// TwinCAT 3 PLC project tcl_BaseClasses
// Title: tcl_BaseClasses
// Company: Red Rock Controls Limited
// Author: Roger Christopher
// ProjectVersion: 1.1.70.0
// Description: ResultAggregate updated to use array of I_ExecutionResult interfaces for transparency during debugging
// ProgramVersion: 3.1.4023.0
// CompilerDefines: VISU_USEPROPERTYINFO
// libraries:
//   Tc2_Standard, * (Beckhoff Automation GmbH)
//   Tc2_System, * (Beckhoff Automation GmbH)
//   Tc2_Utilities, * (Beckhoff Automation GmbH)
//   Tc3_DynamicMemory, * (Beckhoff Automation GmbH)
//   Tc3_EventLogger, * (Beckhoff Automation GmbH)
//   Tc3_Module, * (Beckhoff Automation GmbH)
//   tcl_StringUtils, * (Red Rock Controls Limited)
// project tree:
//   Classes/Change Monitoring/ T_Monitor_INT.TcPOU, T_Monitor_DINT.TcPOU, T_Monitor_Structure.TcPOU
//   Classes/Execution Result Aggregate/ T_ResultAggregate.TcPOU
//   Classes/Execution/Execution/ I_Execution.TcIO, I_ExecutionResult.TcIO, T_Execution.TcPOU, T_ExecutionState.TcDUT
//   Classes/Function Block Wrappers/Classes/ T_Counter.TcPOU, T_FallingEdge.TcPOU, T_MonitoredValue.TcPOU, T_OffTimer.TcPOU, T_OnTimer.TcPOU, T_PulseTimer.TcPOU, T_RisingEdge.TcPOU, T_SquareWave.TcPOU, T_StructureCrcMonitor.TcPOU, T_ValueMonitor.TcPOU, T_ValueMonitorEx.TcPOU
//   Classes/List Of Interfaces/ I_ListItem.TcIO, I_ListOfInterfaces.TcIO, T_ListOfInterfaces.TcPOU
//   Classes/Logger/ I_Logger.TcIO, T_Logger.TcPOU, T_Message.TcPOU
//   Classes/Notifications/List Of Handlers/ T_ListONotificationHandlers.TcPOU
//   Classes/Notifications/Notification Handler/ I_NotificationHandler.TcIO, T_NotificationHandler.TcPOU
//   Classes/Notifications/Notification/ I_Notification.TcIO, T_Notification.TcPOU
//   Classes/Nullable Base Class/ T_NullableBaseClass.TcPOU
//   Classes/Object base class/ T_Object.TcPOU
//   Classes/Stream/ E_ArgTypeId.TcDUT, I_StreamReader.TcIO, I_StreamWriter.TcIO, T_Stream.TcPOU
//   Functions/ F_CompareMem.TcPOU, F_CopyMem.TcPOU, F_DetectOnlineChange.TcPOU, F_DINT_TO_UDINT.TcPOU, F_Dec.TcPOU, F_InLimits.TcPOU, F_ErrorIdToString.TcPOU, F_Inc.TcPOU, F_LinearInterpolation.TcPOU, F_LogError.TcPOU, F_LogMessage.TcPOU, F_LogWarning.TcPOU, F_ReadFlag.TcPOU, F_TaskTime.TcPOU, F_NotEqual.TcPOU, F_Toggle.TcPOU, F_UDINT_TO_DINT.TcPOU, F_ClearMem.TcPOU, F_Equals.TcPOU, F_GetAdsPort.TcPOU
//   / Globals.TcGVL
//   Version/ Global_Version.TcGVL
// real-time tasks:
//   TASK PlcTask: cycle T#10ms, priority 20, ADS port 350
//   TASK PlcTask1: cycle T#10ms, priority 21, ADS port 351

// ---- Classes/Execution/Execution/T_ExecutionState.TcDUT
{attribute 'qualified_only'}
{attribute 'strict'}
TYPE
    T_ExecutionState :
    (
        Ready := 0,
        Starting,
        Busy
    );
END_TYPE

// ---- Classes/Stream/E_ArgTypeId.TcDUT
{attribute 'qualified_only'}
TYPE
    E_ArgTypeId :
    (
        Unknown := 0,
        Type_Blob,
        Type_BOOL,
        Type_BYTE,
        Type_DINT,
        Type_INT,
        Type_LINT,
        Type_LREAL,
        Type_PVOID,
        Type_REAL,
        Type_STRING,
        Type_UDINT,
        Type_UINT,
        Type_ULINT,
        MaxSupportType
    );
END_TYPE

// ---- Globals.TcGVL
VAR_GLOBAL
	DefaultLogger : T_Logger;
END_VAR

// ---- Version/Global_Version.TcGVL
{attribute 'TcGenerated'}
{attribute 'no-analysis'}
{attribute 'linkalways'}
// This function has been automatically generated from the project information.
VAR_GLOBAL CONSTANT
	{attribute 'const_non_replaced'}
	stLibVersion_tcl_BaseClasses : ST_LibVersion := (iMajor := 1, iMinor := 1, iBuild := 70, iRevision := 0, nFlags := 0, sVersion := '1.1.70.0');
END_VAR

// ---- Classes/Execution/Execution/I_Execution.TcIO
INTERFACE I_Execution

METHOD Abort
VAR_INPUT
END_VAR
END_METHOD

PROPERTY Aborted : BOOL
GET
END_GET
END_PROPERTY

PROPERTY Busy : BOOL
GET
END_GET
END_PROPERTY

METHOD Clear
VAR_INPUT
END_VAR
END_METHOD

PROPERTY Done : BOOL
GET
END_GET
END_PROPERTY

PROPERTY Error : BOOL
GET
END_GET
END_PROPERTY

PROPERTY ErrorMsg : T_MaxString
GET
END_GET
END_PROPERTY

PROPERTY Ready : BOOL
GET
END_GET
END_PROPERTY

METHOD Start : I_ExecutionResult;
VAR_INPUT
END_VAR
END_METHOD

PROPERTY Starting : BOOL
GET
END_GET
END_PROPERTY

END_INTERFACE

// ---- Classes/Execution/Execution/I_ExecutionResult.TcIO
INTERFACE I_ExecutionResult EXTENDS I_ListItem // Just exposes the state of the execution object. Usage is "Result := Execution.Start()" so Result can be monitored

METHOD Abort
VAR_INPUT
END_VAR
END_METHOD

PROPERTY Aborted : BOOL
GET
END_GET
END_PROPERTY

PROPERTY Aborting : BOOL
GET
END_GET
END_PROPERTY

PROPERTY Busy : BOOL
GET
END_GET
END_PROPERTY

METHOD Clear
END_METHOD

PROPERTY Done : BOOL
GET
END_GET
END_PROPERTY

PROPERTY Error : BOOL
GET
END_GET
END_PROPERTY

PROPERTY ErrorMsg : T_MaxString
GET
END_GET
END_PROPERTY

PROPERTY Ready : BOOL
GET
END_GET
END_PROPERTY

PROPERTY Starting : BOOL
GET
END_GET
END_PROPERTY

END_INTERFACE

// ---- Classes/List Of Interfaces/I_ListItem.TcIO
INTERFACE I_ListItem EXTENDS __SYSTEM.IQueryInterface

END_INTERFACE

// ---- Classes/List Of Interfaces/I_ListOfInterfaces.TcIO
INTERFACE I_ListOfInterfaces EXTENDS I_ListItem

METHOD AddInterface
VAR_INPUT
    InterfacePointer : I_ListItem;
END_VAR
END_METHOD

PROPERTY Count : DINT
GET
END_GET
END_PROPERTY

METHOD GetInterface : I_ListItem
VAR_INPUT
    Index : DINT;
END_VAR
END_METHOD

END_INTERFACE

// ---- Classes/Logger/I_Logger.TcIO
INTERFACE I_Logger

METHOD LogCritical
VAR_INPUT
	Source	: I_TcSourceInfo;
    Message : T_MaxString;
END_VAR
END_METHOD

METHOD LogDebug
VAR_INPUT
	Source	: I_TcSourceInfo;
    Message : T_MaxString;
END_VAR
END_METHOD

METHOD LogError
VAR_INPUT
	Source	: I_TcSourceInfo;
    Message : T_MaxString;
END_VAR
END_METHOD

METHOD LogInfo
VAR_INPUT
	Source	: I_TcSourceInfo;
    Message : T_MaxString;
END_VAR
END_METHOD

METHOD LogWarning
VAR_INPUT
	Source	: I_TcSourceInfo;
    Message : T_MaxString;
END_VAR
END_METHOD

END_INTERFACE

// ---- Classes/Notifications/Notification Handler/I_NotificationHandler.TcIO
{attribute 'hide'}
INTERFACE I_NotificationHandler EXTENDS __SYSTEM.IQueryInterface

PROPERTY Args : I_StreamReader
GET
END_GET
END_PROPERTY

PROPERTY NotificationCount : DINT
GET
END_GET
END_PROPERTY

METHOD RaiseNotification
VAR_INPUT
    NotificationArgs : I_StreamReader;
END_VAR
END_METHOD

END_INTERFACE

// ---- Classes/Notifications/Notification/I_Notification.TcIO
INTERFACE I_Notification

METHOD AddNotificationHandler : I_Notification
VAR_INPUT
    Handler : I_NotificationHandler;
END_VAR
END_METHOD

PROPERTY Args : I_StreamWriter
GET
END_GET
END_PROPERTY

METHOD ClearNotificationHandlers : I_Notification
VAR_INPUT
END_VAR
END_METHOD

METHOD Raise
END_METHOD

END_INTERFACE

// ---- Classes/Stream/I_StreamReader.TcIO
INTERFACE I_StreamReader

{attribute 'monitoring' := 'call'}
PROPERTY BufferAddress : PVOID
GET
END_GET
END_PROPERTY

METHOD GetNextArgTypeId : E_ArgTypeId
END_METHOD

METHOD Read_BLOB
VAR_INPUT
    BlobToCopyTo : ANY;
END_VAR
END_METHOD

METHOD Read_BOOL : BOOL
END_METHOD

METHOD Read_BYTE : BYTE
END_METHOD

METHOD Read_DATA
VAR_INPUT
    DataAddress : PVOID;
    DataLength  : UDINT;
END_VAR
END_METHOD

METHOD Read_DINT : DINT
END_METHOD

METHOD Read_INT : INT
END_METHOD

METHOD Read_LINT : LINT
END_METHOD

METHOD Read_LREAL : LREAL
END_METHOD

METHOD Read_PVOID : PVOID
END_METHOD

METHOD Read_REAL : REAL
END_METHOD

METHOD Read_STRING : STRING(255)
END_METHOD

METHOD Read_STRUCT
VAR_INPUT
    StructureAddress : PVOID;
    StructureLength  : UDINT;
END_VAR
END_METHOD

METHOD Read_UDINT : UDINT
END_METHOD

METHOD Read_UINT : UINT
END_METHOD

METHOD Read_ULINT : ULINT
END_METHOD

{attribute 'monitoring' := 'call'}
PROPERTY ReadPosition : UDINT
GET
END_GET
END_PROPERTY

METHOD SetReadPosition : I_StreamWriter
VAR_INPUT
    Position : UDINT;
END_VAR
END_METHOD

{attribute 'monitoring' := 'call'}
PROPERTY StreamLength : UDINT
GET
END_GET
END_PROPERTY

{attribute 'monitoring' := 'call'}
PROPERTY WritePosition : UDINT
GET
END_GET
END_PROPERTY

END_INTERFACE

// ---- Classes/Stream/I_StreamWriter.TcIO
INTERFACE I_StreamWriter

METHOD Add_BLOB : I_StreamWriter
VAR_INPUT
    BlobToCopyFrom : ANY;
END_VAR
END_METHOD

METHOD Add_BOOL : I_StreamWriter
VAR_INPUT
    Value : BOOL;
END_VAR
END_METHOD

METHOD Add_BYTE : I_StreamWriter
VAR_INPUT
    Value : BYTE;
END_VAR
END_METHOD

METHOD Add_DATA : I_StreamWriter
VAR_INPUT
    DataAddress : PVOID;
    DataLength  : UDINT;
END_VAR
END_METHOD

METHOD Add_DINT : I_StreamWriter
VAR_INPUT
    Value : DINT;
END_VAR
END_METHOD

METHOD Add_INT : I_StreamWriter
VAR_INPUT
    Value : INT;
END_VAR
END_METHOD

METHOD Add_LINT : I_StreamWriter
VAR_INPUT
    Value : LINT;
END_VAR
END_METHOD

METHOD Add_LREAL : I_StreamWriter
VAR_INPUT
    Value : LREAL;
END_VAR
END_METHOD

METHOD Add_PVOID : I_StreamWriter
VAR_INPUT
    Value : PVOID;
END_VAR
END_METHOD

METHOD Add_REAL : I_StreamWriter
VAR_INPUT
    Value : REAL;
END_VAR
END_METHOD

METHOD Add_STRING : I_StreamWriter
VAR_INPUT
    Value : STRING(255);
END_VAR
END_METHOD

METHOD Add_STRUCT : I_StreamWriter
VAR_INPUT
    StructureAddress : PVOID;
    StructureLength  : UDINT;
END_VAR
END_METHOD

METHOD Add_UDINT : I_StreamWriter
VAR_INPUT
    Value : UDINT;
END_VAR
END_METHOD

METHOD Add_UINT : I_StreamWriter
VAR_INPUT
    Value : UINT;
END_VAR
END_METHOD

METHOD Add_ULINT : I_StreamWriter
VAR_INPUT
    Value : ULINT;
END_VAR
END_METHOD

METHOD AppendBytesFromStream
VAR_INPUT
    StreamToAppend        : I_StreamReader;
    NumberOfBytesToAppend : UDINT;
END_VAR
VAR

END_VAR
END_METHOD

{attribute 'monitoring' := 'call'}
PROPERTY BufferAddress : PVOID
GET
END_GET
END_PROPERTY

METHOD Clear : I_StreamWriter
END_METHOD

METHOD Init
VAR_INPUT
    StreamLength : UDINT;
END_VAR
END_METHOD

{attribute 'monitoring' := 'call'}
PROPERTY ReadPosition : UDINT
GET
END_GET
END_PROPERTY

METHOD SetNextArgTypeId : I_StreamWriter
VAR_INPUT
    Value : E_ArgTypeId;
END_VAR
END_METHOD

METHOD SetReadPosition : I_StreamWriter
VAR_INPUT
    Position : UDINT;
END_VAR
END_METHOD

{attribute 'monitoring' := 'call'}
PROPERTY StreamLength : UDINT
GET
END_GET
END_PROPERTY

{attribute 'monitoring' := 'call'}
PROPERTY WritePosition : UDINT
GET
END_GET
END_PROPERTY

END_INTERFACE

// ---- Classes/Logger/T_Logger.TcPOU
{attribute 'no_explicit_call' := 'do not call this POU directly'}
FUNCTION_BLOCK T_Logger IMPLEMENTS I_Logger
VAR
    DebugMessage    : T_Message;
    InfoMessage     : T_Message;
    WarningMessage  : T_Message;
    ErrorMessage    : T_Message;
    CriticalMessage : T_Message;

END_VAR

METHOD LogCritical
VAR_INPUT
	Source	: I_TcSourceInfo;
	Message	: Tc2_System.T_MaxString;
END_VAR
CriticalMessage.Send(TcEventSeverity.Critical, Source,Message);
END_METHOD

METHOD LogDebug
VAR_INPUT
	Source	: I_TcSourceInfo;
	Message	: Tc2_System.T_MaxString;
END_VAR
DebugMessage.Send(TcEventSeverity.Verbose, Source,Message);
END_METHOD

METHOD LogError
VAR_INPUT
	Source	: I_TcSourceInfo;
	Message	: Tc2_System.T_MaxString;
END_VAR
ErrorMessage.Send(TcEventSeverity.Error, Source,Message);
END_METHOD

METHOD LogInfo
VAR_INPUT
	Source	: I_TcSourceInfo;
	Message	: Tc2_System.T_MaxString;
END_VAR
InfoMessage.Send(TcEventSeverity.Info, Source,Message);
END_METHOD

METHOD LogWarning
VAR_INPUT
	Source	: I_TcSourceInfo;
	Message	: Tc2_System.T_MaxString;
END_VAR
WarningMessage.Send(TcEventSeverity.Warning, Source,Message);
END_METHOD

END_FUNCTION_BLOCK

// ---- Classes/Logger/T_Message.TcPOU
FUNCTION_BLOCK T_Message
VAR
    Msg        : FB_TcMessage;
END_VAR

METHOD Send
VAR_INPUT
    Severity : TcEventSeverity;
    Source   : I_TcSourceInfo;
    Message  : Tc2_System.T_MaxString;
END_VAR
VAR
    Result : HRESULT;
END_VAR
CASE Severity OF 
	TcEventSeverity.Critical:
		Result := Msg.CreateEx(TC_EVENTS.PLC_Exceptions.LogCritical, Source);
		
	TcEventSeverity.Error:
		Result := Msg.CreateEx(TC_EVENTS.PLC_Exceptions.LogError, Source);
		
	TcEventSeverity.Warning:
		Result := Msg.CreateEx(TC_EVENTS.PLC_Exceptions.LogWarning, Source);
		
	TcEventSeverity.Info:
		Result := Msg.CreateEx(TC_EVENTS.PLC_Exceptions.LogInfo, Source);
		
	TcEventSeverity.Verbose:
		Result := Msg.CreateEx(TC_EVENTS.PLC_Exceptions.LogDebug, Source);
		
END_CASE

IF Result = S_OK THEN
	Msg.ipArguments.Clear().AddString(Message);
    Msg.Send(0);
	Msg.Release();
ELSE
    F_LogError(Source := 'Logger', 'Failed to create EventLogger.Message instance');
END_IF
END_METHOD

END_FUNCTION_BLOCK

// ---- Functions/F_LogError.TcPOU
FUNCTION F_LogError
VAR_INPUT
    Source  : T_MaxString;
    Message : T_MaxString;
END_VAR
VAR_STAT
    LastMessage        : T_MaxString;
    RepeatMessageCount : UDINT;
END_VAR

IF Message = LastMessage THEN
    F_Inc(RepeatMessageCount);
ELSE
    RepeatMessageCount := 0;
    LastMessage        := Message;
END_IF

IF RepeatMessageCount < 10 THEN // Avoid flooding the Error List...
    ADSLOGSTR(msgCtrlMask := ADSLOG_MSGTYPE_STRING OR ADSLOG_MSGTYPE_ERROR OR ADSLOG_MSGTYPE_LOG,
              msgFmtStr   := CONCAT(Source, ' : %s'),
              strArg      := Message);
END_IF

IF RepeatMessageCount = 10 THEN
    ADSLOGSTR(msgCtrlMask := ADSLOG_MSGTYPE_STRING OR ADSLOG_MSGTYPE_ERROR OR ADSLOG_MSGTYPE_LOG,
              msgFmtStr   := 'Log Errors suspended - too many identical messages!',
              strArg      := '');
END_IF

END_FUNCTION

// ---- Functions/F_Inc.TcPOU
FUNCTION F_Inc : BOOL
VAR_INPUT
    in : ANY_INT;
END_VAR
VAR
    pSINT  : POINTER TO SINT;
    pINT   : POINTER TO INT;
    pDINT  : POINTER TO DINT;
    pLINT  : POINTER TO LINT;
    pUSINT : POINTER TO USINT;
    pUINT  : POINTER TO UINT;
    pUDINT : POINTER TO UDINT;
    pULINT : POINTER TO ULINT;
    pBYTE  : POINTER TO BYTE;
    pWORD  : POINTER TO WORD;
    pDWORD : POINTER TO DWORD;
END_VAR

CASE in.TypeClass OF
    __SYSTEM.TYPE_CLASS.TYPE_SINT:
        pSINT  := in.pValue;
        pSint^ := pSint^ + 1;

    __SYSTEM.TYPE_CLASS.TYPE_INT:
        pINT  := in.pValue;
        pINT^ := pINT^ + 1;

    __SYSTEM.TYPE_CLASS.TYPE_DINT:
        pDINT  := in.pValue;
        pDINT^ := pDINT^ + 1;

    __SYSTEM.TYPE_CLASS.TYPE_LINT:
        pLINT  := in.pValue;
        pLINT^ := pLINT^ + 1;

    __SYSTEM.TYPE_CLASS.TYPE_USINT:
        pUSINT  := in.pValue;
        pUSINT^ := pUSINT^ + 1;

    __SYSTEM.TYPE_CLASS.TYPE_UINT:
        pUINT  := in.pValue;
        pUINT^ := pUINT^ + 1;

    __SYSTEM.TYPE_CLASS.TYPE_UDINT:
        pUDINT  := in.pValue;
        pUDINT^ := pUDINT^ + 1;

    __SYSTEM.TYPE_CLASS.TYPE_ULINT:
        pULINT  := in.pValue;
        pULINT^ := pULINT^ + 1;
		
    __SYSTEM.TYPE_CLASS.TYPE_BYTE:
        pBYTE  := in.pValue;
        pBYTE^ := pBYTE^ + 1;
		
    __SYSTEM.TYPE_CLASS.TYPE_WORD:
        pWORD  := in.pValue;
        pWORD^ := pWORD^ + 1;
		
    __SYSTEM.TYPE_CLASS.TYPE_DWORD:
        pDWORD  := in.pValue;
        pDWORD^ := pDWORD^ + 1;
		
		
END_CASE

END_FUNCTION

// ---- Classes/Change Monitoring/T_Monitor_INT.TcPOU
{attribute 'no_explicit_call':= 'do not call this POU directly'}
FUNCTION_BLOCK T_Monitor_INT
VAR
    _CurrentValue  : INT := UnlikelyValue; 
    _Changed       : BOOL;
END_VAR
VAR CONSTANT
	UnlikelyValue : INT := 12345;
END_VAR

PROPERTY Changed : BOOL
GET
Changed := _Changed;
END_GET
END_PROPERTY

METHOD CyclicUpdate : BOOL
VAR_INPUT
    Value : INT;
END_VAR
_Changed      := Value <> _CurrentValue;
_CurrentValue := Value;
CyclicUpdate  := _Changed;
END_METHOD

METHOD Reset
_CurrentValue := UnlikelyValue;
_Changed      := FALSE;
END_METHOD

END_FUNCTION_BLOCK

// ---- Classes/Change Monitoring/T_Monitor_DINT.TcPOU
{attribute 'no_explicit_call':= 'do not call this POU directly'}
FUNCTION_BLOCK T_Monitor_DINT
VAR
    _CurrentValue  : DINT := UnlikelyValue; 
    _Changed       : BOOL;
END_VAR
VAR CONSTANT
	UnlikelyValue : DINT := 123456789;
END_VAR

PROPERTY Changed : BOOL
GET
Changed := _Changed;
END_GET
END_PROPERTY

METHOD CyclicUpdate : BOOL
VAR_INPUT
    Value : DINT;
END_VAR
_Changed      := Value <> _CurrentValue;
_CurrentValue := Value;
CyclicUpdate  := _Changed;
END_METHOD

METHOD Reset
_CurrentValue := UnlikelyValue;
_Changed      := FALSE;
END_METHOD

END_FUNCTION_BLOCK

// ---- Classes/Change Monitoring/T_Monitor_Structure.TcPOU
{attribute 'no_explicit_call':= 'do not call this POU directly'}
FUNCTION_BLOCK T_Monitor_Structure
VAR
    _Changed   : BOOL;
    Stored_CRC : WORD := 16#FFFF;
END_VAR

PROPERTY Changed : BOOL
GET
Changed := _Changed;
END_GET
END_PROPERTY

METHOD CyclicUpdate : BOOL
VAR_INPUT
    StructureAddress : PVOID;
	StructureLength  : UDINT;
END_VAR
VAR
    CRC : WORD;
END_VAR
CRC := F_DATA_TO_CRC16_CCITT(pData  := StructureAddress,
                             cbData := StructureLength,
                             crc    := 0);
_Changed := (CRC <> Stored_CRC);
IF Changed THEN
    Stored_CRC := CRC;
END_IF
CyclicUpdate := _Changed;
END_METHOD

METHOD Reset
VAR_INPUT
END_VAR
Stored_CRC := 16#FFFF;
_Changed   := FALSE;
END_METHOD

END_FUNCTION_BLOCK

// ---- Classes/Execution Result Aggregate/T_ResultAggregate.TcPOU
FUNCTION_BLOCK T_ResultAggregate IMPLEMENTS I_ExecutionResult
VAR
	Results : ARRAY[0..ResultsUpperBound] OF I_ExecutionResult;
	Count   : UINT;
END_VAR
VAR CONSTANT
	ResultsUpperBound : UINT := 99;
END_VAR

METHOD Abort
VAR
    i      : DINT;
    Result : I_ExecutionResult;
    IP     : I_ListItem;
END_VAR
IF Count > 0 THEN
	FOR i := 0 TO Count - 1 DO
		Result := Results[i];
		IF Result <> 0 THEN
            Result.Abort(); 
        END_IF
    END_FOR
END_IF
END_METHOD

PROPERTY Aborted : BOOL
GET
VAR
    i      : UINT;
    Result : I_ExecutionResult;
END_VAR
Aborted := TRUE;
IF Count > 0 THEN
	FOR i := 0 TO Count - 1 DO
		Result := Results[i];
		IF Result <> 0 THEN
			Aborted := Aborted AND Result.Aborted; // Done if all result.aborted
		END_IF
	END_FOR
END_IF
END_GET
END_PROPERTY

PROPERTY Aborting : BOOL
GET
VAR
    i      : DINT;
    Result : I_ExecutionResult;
    IP     : I_ListItem;
END_VAR
Aborting := FALSE;
IF Count > 0 THEN
	FOR i := 0 TO Count - 1 DO
		Result := Results[i];
		IF Result <> 0 THEN
            Aborting := Aborting OR Result.Aborting; // Busy if any result.aborting
        END_IF
    END_FOR
END_IF
END_GET
END_PROPERTY

METHOD AddResult : BOOL
VAR_INPUT
	Result : I_ExecutionResult;
END_VAR
IF Count <= ResultsUpperBound THEN
	Results[Count] := Result;
	F_Inc(Count);
	AddResult := TRUE;
END_IF
END_METHOD

PROPERTY Busy : BOOL
GET
VAR
    i      : DINT;
    Result : I_ExecutionResult;
    IP     : I_ListItem;
END_VAR
Busy := FALSE;
IF Count > 0 THEN
	FOR i := 0 TO Count - 1 DO
		Result := Results[i];
		IF Result <> 0 THEN
            Busy := Busy OR Result.Busy; // Busy if any result.busy
        END_IF
    END_FOR
END_IF
END_GET
END_PROPERTY

METHOD Clear
VAR
    i      : UINT;
    Result : I_ExecutionResult;
END_VAR
IF Count > 0 THEN
    FOR i := 0 TO Count - 1 DO
		Result := Results[i];
		IF Result <> 0 THEN
			Result.Clear(); 
		END_IF
	END_FOR
END_IF

F_ClearMem(Results);
Count := 0;
END_METHOD

PROPERTY Done : BOOL
GET
VAR
    i      : DINT;
    Result : I_ExecutionResult;
    IP     : I_ListItem;
END_VAR
Done := TRUE;
IF Count > 0 THEN
	FOR i := 0 TO Count - 1 DO
		Result := Results[i];
		IF Result <> 0 THEN
			Done := Done AND Result.Done; // Done if all result.done
		END_IF
	END_FOR
END_IF
END_GET
END_PROPERTY

PROPERTY Error : BOOL
GET
VAR
    i      : DINT;
    Result : I_ExecutionResult;
    IP     : I_ListItem;
END_VAR
Error := FALSE;
IF Count > 0 THEN
	FOR i := 0 TO Count - 1 DO
		Result := Results[i];
		IF Result <> 0 THEN
			Error := Error OR Result.Error; // Error if any result.error
		END_IF
	END_FOR
END_IF
END_GET
END_PROPERTY

PROPERTY ErrorMsg : Tc2_System.T_MaxString
GET
VAR
    i      : DINT;
    Result : I_ExecutionResult;
    IP     : I_ListItem;
END_VAR
ErrorMsg := '';
IF Count > 0 THEN
	FOR i := 0 TO Count - 1 DO
		Result := Results[i];
		IF Result <> 0 THEN
			IF Result.Error THEN
				ErrorMsg := Result.ErrorMsg;
				RETURN;
			END_IF
		END_IF
	END_FOR
END_IF
END_GET
END_PROPERTY

PROPERTY Ready : BOOL
GET
VAR
    i      : DINT;
    Result : I_ExecutionResult;
    IP     : I_ListItem;
END_VAR
Ready := TRUE;
IF Count > 0 THEN
	FOR i := 0 TO Count - 1 DO
		Result := Results[i];
		IF Result <> 0 THEN
            Ready := Ready AND Result.Ready; // Ready if all result.ready
        END_IF
    END_FOR
END_IF
END_GET
END_PROPERTY

PROPERTY ResultCount : DINT
GET
ResultCount := Count;
END_GET
END_PROPERTY

PROPERTY Starting : BOOL
GET
VAR
    i      : DINT;
    Result : I_ExecutionResult;
    IP     : I_ListItem;
END_VAR
Starting := FALSE;
IF Count > 0 THEN
	FOR i := 0 TO Count - 1 DO
		Result := Results[i];
		IF Result <> 0 THEN
            Starting := Starting OR Result.Starting; // Starting if any result.starting
        END_IF
    END_FOR
END_IF
END_GET
END_PROPERTY

END_FUNCTION_BLOCK

// ---- Functions/F_ClearMem.TcPOU
FUNCTION F_ClearMem : BOOL
VAR_INPUT
    Data : ANY;
END_VAR
VAR
END_VAR

MEMSET(destAddr := Data.pValue,
       fillByte := 0,
       n        := DINT_TO_UDINT(Data.diSize));

END_FUNCTION

// ---- Classes/Execution/Execution/T_Execution.TcPOU
// Class for handling communications between a client requesting a service 
// and a server providing the service

FUNCTION_BLOCK T_Execution EXTENDS T_Object IMPLEMENTS I_Execution, I_ExecutionResult
VAR
    _State    : T_ExecutionState;
    _Done     : BOOL;
    _Error    : BOOL;
    _Aborted  : BOOL;
    _ErrorMsg : T_MaxString;
    _Aborting : BOOL;
END_VAR

METHOD Abort
_Aborting := TRUE;
END_METHOD

PROPERTY Aborted : BOOL
GET
Aborted := _Aborted;
END_GET
END_PROPERTY

PROPERTY Aborting : BOOL
GET
Aborting := _Aborting;
END_GET
END_PROPERTY

PROPERTY Busy : BOOL
GET
Busy := _State = T_ExecutionState.Busy;
END_GET
END_PROPERTY

METHOD Clear
_Done     := FALSE;
_Aborted  := FALSE;
_Error    := FALSE;
_Aborting := FALSE;
_ErrorMsg := '';
_State    := T_ExecutionState.Ready;
END_METHOD

PROPERTY Done : BOOL
GET
Done := _Done;
END_GET
END_PROPERTY

PROPERTY Error : BOOL
GET
Error := _Error;
END_GET
END_PROPERTY

PROPERTY ErrorMsg : T_MaxString
GET
ErrorMsg := _ErrorMsg;
END_GET
END_PROPERTY

METHOD FB_init : BOOL
VAR_INPUT
	bInitRetains : BOOL; // if TRUE, the retain variables are initialized (warm start / cold start)
	bInCopyCode : BOOL;  // if TRUE, the instance afterwards gets moved into the copy code (online change)
END_VAR
_Source.sName := 'Execution';
END_METHOD

PROPERTY Name : T_MaxString
GET
Name := SUPER^._Name;
END_GET
END_PROPERTY

PROPERTY Ready : BOOL
GET
Ready := _State = T_ExecutionState.Ready;
END_GET
END_PROPERTY

METHOD SetAborted
_Aborting := FALSE;
_Done     := FALSE;
_Error    := FALSE;

IF _State <> T_ExecutionState.Ready THEN
    _Aborted  := TRUE;
    _ErrorMsg := F_FormatStringEx1('%s - Execution aborted',SUPER^._Name);
    _State    := T_ExecutionState.Ready;
	
	_Message.CreateEx(TC_EVENTS.PLC_Exceptions.LogWarning,_Source);
	_Message.ipArguments.AddString(_ErrorMsg);
	_Message.Send(0);
	_Message.Release();
END_IF
END_METHOD

METHOD SetBusy
VAR_INPUT
END_VAR
IF _State = T_ExecutionState.Starting THEN
    _State := T_ExecutionState.Busy;
END_IF
END_METHOD

METHOD SetDone
VAR_INPUT
END_VAR
IF _State = T_ExecutionState.Starting OR _State = T_ExecutionState.Busy THEN
    _Error    := FALSE;
    _ErrorMsg := '';
    _Aborted  := FALSE;
    _Done     := TRUE;
    _State    := T_ExecutionState.Ready;
END_IF
END_METHOD

METHOD SetError
VAR_INPUT
    ErrorMsg : T_MaxString;
END_VAR
VAR_INST
	fullMessage : T_MaxString;
END_VAR
_Error    := TRUE;
_Aborted  := FALSE;
_Done     := FALSE;
_ErrorMsg := ErrorMsg;
_State    := T_ExecutionState.Ready;

fullMessage := F_FormatStringEx2('%s - %s', _Name, ErrorMsg);
_Message.CreateEx(TC_EVENTS.PLC_Exceptions.LogError, _Source);
_Message.ipArguments.AddString(fullMessage);
_Message.Send(0);
_Message.Release();
END_METHOD

METHOD Start : I_ExecutionResult
VAR_INPUT
END_VAR
IF _State = T_ExecutionState.Ready THEN
    _Done     := FALSE;
    _Aborted  := FALSE;
    _Error    := FALSE;
    _ErrorMsg := '';
    _State := T_ExecutionState.Starting;
	
ELSIF _State = T_ExecutionState.Busy THEN
    SetError('Start requested while already busy');
	
ELSIF _State = T_ExecutionState.Starting THEN
    SetError('Start requested while already starting');
	
ELSIF _Aborting THEN
    SetError('Start requested while aborting');
	
ELSE
    SetError('Start requested while not ready');
END_IF

Start := THIS^;
END_METHOD

PROPERTY Starting : BOOL
GET
Starting := _State = T_ExecutionState.Starting;
END_GET
END_PROPERTY

PROPERTY State : T_ExecutionState
GET
State := _State;
END_GET
END_PROPERTY

END_FUNCTION_BLOCK

// ---- Classes/Object base class/T_Object.TcPOU
{attribute 'reflection'}
FUNCTION_BLOCK T_Object
VAR
    {attribute 'instance-path'}
    {attribute 'no_init'}
    _Name     : T_MaxString; // Automatically initialised with the full name of the instance
    _Project  : T_MaxString;
    _Solution : T_MaxString;

    _Source  : FB_TcSourceInfo;
    _Message : FB_TcMessage;
END_VAR

METHOD FB_init : BOOL
VAR_INPUT
    bInitRetains : BOOL; // if TRUE, the retain variables are initialized (warm start / cold start)
    bInCopyCode  : BOOL; // if TRUE, the instance afterwards gets moved into the copy code (online change)
END_VAR
VAR
    StringSplitter : T_StringSplitter;
END_VAR
StringSplitter.Init(Str    := _Name,
                    Delim1 := '.',
                    Delim2 := '');

_Solution := StringSplitter.GetNext();
_Project  := StringSplitter.GetNext();
_Name     := StringSplitter.GetRemainder();

_Source.sName := _Name;
END_METHOD

END_FUNCTION_BLOCK

// ---- Classes/Function Block Wrappers/Classes/T_Counter.TcPOU
FUNCTION_BLOCK T_Counter
VAR
    Count : DINT;
END_VAR

METHOD Dec : DINT
VAR_INPUT
END_VAR
Count := Count - 1;
Dec   := Count;
END_METHOD

METHOD Inc : DINT
VAR_INPUT
END_VAR
Count := Count + 1;
Inc   := Count;
END_METHOD

METHOD Init
VAR_INPUT
    Value : DINT;
END_VAR
Count := Value;
END_METHOD

METHOD Reset
VAR_INPUT
END_VAR
Count := 0;
END_METHOD

PROPERTY Value : DINT
GET
Value := Count;
END_GET
END_PROPERTY

PROPERTY ValueAsTArg : T_Arg
GET
ValueAsTArg := F_DINT(Count);
END_GET
END_PROPERTY

END_FUNCTION_BLOCK

// ---- Classes/Function Block Wrappers/Classes/T_FallingEdge.TcPOU
FUNCTION_BLOCK T_FallingEdge
VAR
    F_TRIG1 : F_TRIG;
END_VAR

PROPERTY EdgeDetected : BOOL
GET
EdgeDetected := F_TRIG1.Q;
END_GET
END_PROPERTY

METHOD Test : BOOL
VAR_INPUT
    Value : BOOL;
END_VAR
F_TRIG1(CLK := Value);
Test := F_TRIG1.Q;
END_METHOD

END_FUNCTION_BLOCK

// ---- Classes/Function Block Wrappers/Classes/T_MonitoredValue.TcPOU
FUNCTION_BLOCK T_MonitoredValue
VAR_INPUT
END_VAR
VAR_OUTPUT
END_VAR
VAR
    _Value   : LREAL;
    _Changed : BOOL;
	_ChangeThreshold : LREAL;
END_VAR

PROPERTY Changed : BOOL
GET
Changed := _Changed;
END_GET
END_PROPERTY

METHOD FB_init : BOOL
VAR_INPUT
    bInitRetains    : BOOL; // if TRUE, the retain variables are initialized (warm start / cold start)
    bInCopyCode     : BOOL; // if TRUE, the instance afterwards gets moved into the copy code (online change)
    ChangeThreshold : LREAL;
END_VAR
THIS^._ChangeThreshold := ChangeThreshold;
END_METHOD

METHOD Read : LREAL
VAR_INPUT
END_VAR
Read     := _Value;
_Changed := FALSE;
END_METHOD

METHOD Update
VAR_INPUT
	Value : LREAL;
END_VAR
IF ABS(Value - _Value) > _ChangeThreshold THEN
	_Value := Value;
	_Changed := TRUE;
END_IF
END_METHOD

END_FUNCTION_BLOCK

// ---- Classes/Function Block Wrappers/Classes/T_OffTimer.TcPOU
FUNCTION_BLOCK T_OffTimer
VAR
    TOF1 : TOF;
END_VAR

METHOD Delay : BOOL
VAR_INPUT
    In : BOOL;
END_VAR
TOF1(IN := In);
Delay := TOF1.Q;
END_METHOD

METHOD FB_init : BOOL
VAR_INPUT
    bInitRetains : BOOL;  // if TRUE, the retain variables are initialized (warm start / cold start)
    bInCopyCode  : BOOL;  // if TRUE, the instance afterwards gets moved into the copy code (online change)
    PresetTime   : LREAL; // seconds
END_VAR
TOF1.PT := LREAL_TO_TIME(PresetTime * 1000);
END_METHOD

PROPERTY OutputState : BOOL
GET
OutputState := TOF1.Q;
END_GET
END_PROPERTY

PROPERTY PresetTime : LREAL
GET
PresetTime := TIME_TO_LREAL(TOF1.PT) / 1000.0; // in seconds
END_GET
SET
TOF1.PT := LREAL_TO_TIME(PresetTime * 1000);
END_SET
END_PROPERTY

END_FUNCTION_BLOCK

// ---- Classes/Function Block Wrappers/Classes/T_OnTimer.TcPOU
FUNCTION_BLOCK T_OnTimer
VAR
    TON1 : TON;
END_VAR

METHOD Clock : BOOL
TON1(IN := TRUE);
Clock := TON1.Q;
IF Clock THEN
    TON1(IN := FALSE);
END_IF
END_METHOD

METHOD Delay : BOOL
VAR_INPUT
    In : BOOL;
END_VAR
TON1(IN := In);
Delay := TON1.Q;
END_METHOD

PROPERTY ElapsedTime : LREAL
GET
ElapsedTime := TIME_TO_LREAL(TON1.ET) / 1000.0; // in seconds
END_GET
END_PROPERTY

METHOD FB_init : BOOL
VAR_INPUT
    bInitRetains : BOOL;  // if TRUE, the retain variables are initialized (warm start / cold start)
    bInCopyCode  : BOOL;  // if TRUE, the instance afterwards gets moved into the copy code (online change)
    PresetTime   : LREAL; // seconds
END_VAR
TON1.PT := LREAL_TO_TIME(PresetTime * 1000);
END_METHOD

PROPERTY OutputState : BOOL
GET
OutputState := TON1.Q;
END_GET
END_PROPERTY

PROPERTY PresetTime : LREAL
GET
PresetTime := TIME_TO_LREAL(TON1.PT) / 1000.0; // in seconds
END_GET
SET
TON1.PT := LREAL_TO_TIME(PresetTime * 1000);
END_SET
END_PROPERTY

METHOD Reset
TON1(IN := FALSE);
END_METHOD

METHOD Run : BOOL
TON1(IN := TRUE);
Run := TON1.Q;
END_METHOD

END_FUNCTION_BLOCK

// ---- Classes/Function Block Wrappers/Classes/T_PulseTimer.TcPOU
FUNCTION_BLOCK T_PulseTimer
VAR
    TP1 : TP;
END_VAR

METHOD FB_init : BOOL
VAR_INPUT
    bInitRetains : BOOL;  // if TRUE, the retain variables are initialized (warm start / cold start)
    bInCopyCode  : BOOL;  // if TRUE, the instance afterwards gets moved into the copy code (online change)
    PresetTime   : LREAL; // seconds
END_VAR
TP1.PT := LREAL_TO_TIME(PresetTime * 1000);
END_METHOD

PROPERTY OutputState : BOOL
GET
OutputState := TP1.Q;
END_GET
END_PROPERTY

PROPERTY PresetTime : LREAL
GET
PresetTime := TIME_TO_LREAL(TP1.PT) / 1000.0; // in seconds
END_GET
SET
TP1.PT := LREAL_TO_TIME(PresetTime * 1000);
END_SET
END_PROPERTY

METHOD Pulse : BOOL
VAR_INPUT
    In : BOOL;
END_VAR
TP1(IN := In);
Pulse := TP1.Q;
END_METHOD

METHOD Reset
TP1(IN := FALSE);
END_METHOD

METHOD Run : BOOL
TP1(IN := TRUE);
Run := TP1.Q;
END_METHOD

END_FUNCTION_BLOCK

// ---- Classes/Function Block Wrappers/Classes/T_RisingEdge.TcPOU
FUNCTION_BLOCK T_RisingEdge
VAR
    R_TRIG1 : R_TRIG;
END_VAR

PROPERTY EdgeDetected : BOOL
GET
EdgeDetected := R_TRIG1.Q;
END_GET
END_PROPERTY

METHOD Test : BOOL
VAR_INPUT
    Value : BOOL;
END_VAR
R_TRIG1(CLK := Value);
Test := R_TRIG1.Q;
END_METHOD

END_FUNCTION_BLOCK

// ---- Classes/Function Block Wrappers/Classes/T_SquareWave.TcPOU
FUNCTION_BLOCK T_SquareWave
VAR
    OnTimer_Mark  : T_OnTimer(PresetTime := 0.5);
    OnTimer_Space : T_Ontimer(PresetTime := 0.5);
    _Output       : BOOL;
END_VAR

IF OnTimer_Mark.Delay(_Output) THEN
    _Output := FALSE;
END_IF

IF OnTimer_Space.Delay(NOT _Output) THEN
    _Output := TRUE;
END_IF

METHOD FB_init : BOOL
VAR_INPUT
    bInitRetains  : BOOL; // if TRUE, the retain variables are initialized (warm start / cold start)
    bInCopyCode   : BOOL; // if TRUE, the instance afterwards gets moved into the copy code (online change)
    MarkDuration  : LREAL;
    SpaceDuration : LREAL;
END_VAR
OnTimer_Mark.PresetTime  := MarkDuration;
OnTimer_Space.PresetTime := SpaceDuration;
END_METHOD

PROPERTY Output : BOOL
GET
Output := _Output;
END_GET
END_PROPERTY

END_FUNCTION_BLOCK

// ---- Classes/Function Block Wrappers/Classes/T_StructureCrcMonitor.TcPOU
{attribute 'no_explicit_call':= 'do not call this POU directly'}
FUNCTION_BLOCK T_StructureCrcMonitor 
VAR
    _Changed   : BOOL;
    Stored_CRC : WORD := 16#FFFF;
END_VAR

PROPERTY Changed : BOOL
GET
Changed := _Changed;
END_GET
END_PROPERTY

METHOD Reset
VAR_INPUT
END_VAR
Stored_CRC := 16#FFFF;
END_METHOD

METHOD Test : BOOL 
VAR_INPUT
    Structure : ANY;
END_VAR
VAR
    CRC : WORD;
END_VAR
CRC := F_DATA_TO_CRC16_CCITT(pData  := Structure.pValue,
                             cbData := DINT_TO_UDINT(Structure.diSize),
                             crc    := 0);

_Changed := (CRC <> Stored_CRC);

IF Changed THEN
    Stored_CRC := CRC;
END_IF

Test := _Changed;
END_METHOD

END_FUNCTION_BLOCK

// ---- Classes/Function Block Wrappers/Classes/T_ValueMonitor.TcPOU
{attribute 'no_explicit_call':= 'do not call this POU directly'}
FUNCTION_BLOCK T_ValueMonitor 
VAR
    _CurrentValue  : INT := -1;
    _PreviousValue : INT;
    _Changed       : BOOL;
END_VAR

PROPERTY Changed : BOOL
GET
Changed := _Changed;
END_GET
END_PROPERTY

PROPERTY CurrentValue : INT
GET
CurrentValue := _CurrentValue;
END_GET
END_PROPERTY

PROPERTY PreviousValue : INT
GET
PreviousValue := _PreviousValue;
END_GET
END_PROPERTY

METHOD Reset
VAR_INPUT
END_VAR
_CurrentValue  := 0;
_PreviousValue := 0;
END_METHOD

METHOD Test : BOOL
VAR_INPUT
    Value : INT;
END_VAR
_Changed       := Value <> _CurrentValue;
_PreviousValue := _CurrentValue;
_CurrentValue  := Value;

Test := _Changed;
END_METHOD

END_FUNCTION_BLOCK

// ---- Classes/Function Block Wrappers/Classes/T_ValueMonitorEx.TcPOU
{attribute 'no_explicit_call':= 'do not call this POU directly'}
FUNCTION_BLOCK T_ValueMonitorEx
VAR
    _Changed    : BOOL;
    StoredValue : ARRAY[0..7] OF BYTE;
END_VAR

PROPERTY Changed : BOOL
GET
Changed := _Changed;
END_GET
END_PROPERTY

METHOD Reset
VAR_INPUT
END_VAR
MEMSET(destAddr := ADR(StoredValue),
       fillByte := 16#00,
       n        := SIZEOF(StoredValue));
END_METHOD

METHOD Test : BOOL;
VAR_INPUT
    Value : ANY_NUM;
END_VAR
_Changed := 0 <>
            MEMCMP(pBuf1 := Value.pValue,
                   pBuf2 := ADR(StoredValue),
                   n     := DINT_TO_UDINT(Value.diSize));

IF _Changed THEN
    MEMCPY(destAddr := ADR(StoredValue),
           srcAddr  := Value.pValue,
           n        := DINT_TO_UDINT(Value.diSize));
END_IF

Test := _Changed;
END_METHOD

END_FUNCTION_BLOCK

// ---- Classes/List Of Interfaces/T_ListOfInterfaces.TcPOU
FUNCTION_BLOCK T_ListOfInterfaces IMPLEMENTS I_ListOfInterfaces
VAR
    {attribute 'analysis' := '-33'} // inhibit unused variable warning
    DynamicMemoryManager : FB_DynMem_Manager;
    Buffer               : FB_DynMem_Buffer(ipMemMan := DynamicMemoryManager);
    pInterface           : POINTER TO I_ListItem;
    _Count               : DINT;
    Capacity             : DINT;
END_VAR

METHOD AddInterface
VAR_INPUT
    InterfacePointer : I_ListItem;
END_VAR
IF _Count = Capacity THEN
    Capacity := Capacity * 2;
    Buffer.Resize(nSize     := DINT_TO_UDINT(Capacity) * SIZEOF(PVOID),
                  bPreserve := TRUE,
                  bReset    := FALSE);

    pInterface := Buffer.pBuffer;
END_IF

IF pInterface <> 0 THEN
    pInterface[_Count] := InterfacePointer;
    _Count             := _Count + 1;
END_IF
END_METHOD

METHOD Clear
VAR_INPUT
END_VAR
IF pInterface = 0 THEN
    // Buffer was not allocated during Fb_init. Try again...
    Buffer.CreateBuffer(nSize  := DINT_TO_UDINT(Capacity) * SIZEOF(PVOID),
                        bReset := TRUE);
END_IF

Buffer.Clear();
_Count := 0;
END_METHOD

PROPERTY Count : DINT
GET
Count := _Count;
END_GET
END_PROPERTY

METHOD FB_exit : BOOL
VAR_INPUT
    bInCopyCode : BOOL; // if TRUE, the exit method is called for exiting an instance that is copied afterwards (online change).
END_VAR
IF NOT bInCopyCode THEN
    Buffer.DeleteBuffer();
    pInterface := 0;
END_IF
END_METHOD

METHOD FB_init : BOOL
VAR_INPUT
    bInitRetains : BOOL; // if TRUE, the retain variables are initialized (warm start / cold start)
    bInCopyCode  : BOOL; // if TRUE, the instance afterwards gets moved into the copy code (online change)
    Capacity     : DINT;
END_VAR
Buffer.CreateBuffer(nSize  := DINT_TO_UDINT(Capacity) * SIZEOF(PVOID),
                    bReset := TRUE);

pInterface := Buffer.pBuffer;

THIS^.Capacity := Capacity;
END_METHOD

METHOD GetInterface : I_ListItem
VAR_INPUT
    Index : DINT;
END_VAR
IF Index < _Count AND Index >= 0 THEN
    GetInterface := pInterface[Index];
END_IF
END_METHOD

END_FUNCTION_BLOCK

// ---- Classes/Notifications/List Of Handlers/T_ListONotificationHandlers.TcPOU
{attribute 'hide'}
FUNCTION_BLOCK T_ListONotificationHandlers
VAR
    Buffer               : FB_DynMem_Buffer(ipMemMan := DynamicMemoryManager);
    DynamicMemoryManager : FB_DynMem_Manager;

    pHandler     : POINTER TO I_NotificationHandler;
    HandlerCount : UDINT;
    Capacity     : UDINT;
END_VAR

METHOD AddHandler
VAR_INPUT
    Handler : I_NotificationHandler;
END_VAR
IF pHandler = 0 THEN // Need  to initialise list of handlers - after online change?
    FB_Init(bInitRetains := FALSE,
            bInCopyCode  := FALSE,
            Capacity     := THIS^.Capacity);

END_IF

IF HandlerInList(Handler) THEN
    RETURN;
END_IF

IF Count = Capacity THEN
    Capacity := Capacity * 2;
    Buffer.Resize(nSize     := Capacity * SIZEOF(PVOID),
                  bPreserve := TRUE,
                  bReset    := FALSE);

    pHandler := Buffer.pBuffer;
END_IF

pHandler[HandlerCount] := Handler;
HandlerCount           := HandlerCount + 1;
END_METHOD

METHOD Clear
VAR_INPUT
END_VAR
Buffer.Clear();
HandlerCount := 0;
END_METHOD

PROPERTY Count : UDINT
GET
Count := HandlerCount;
END_GET
END_PROPERTY

METHOD FB_exit : BOOL
VAR_INPUT
    bInCopyCode : BOOL; // if TRUE, the exit method is called for exiting an instance that is copied afterwards (online change).
END_VAR
IF NOT bInCopyCode THEN
    Buffer.DeleteBuffer();
    pHandler := 0;
END_IF
END_METHOD

METHOD FB_init : BOOL
VAR_INPUT
    bInitRetains : BOOL; // if TRUE, the retain variables are initialized (warm start / cold start)
    bInCopyCode  : BOOL; // if TRUE, the instance afterwards gets moved into the copy code (online change)
    Capacity     : UDINT;
END_VAR
Buffer.CreateBuffer(nSize  := Capacity * SIZEOF(PVOID),
                    bReset := TRUE);

pHandler       := Buffer.pBuffer;
THIS^.Capacity := Capacity;
END_METHOD

METHOD GetHandler : I_NotificationHandler
VAR_INPUT
    Index : UDINT;
END_VAR
IF Index < HandlerCount AND Index >= 0 THEN
    GetHandler := pHandler[Index];
END_IF
END_METHOD

METHOD HandlerInList : BOOL
VAR_INPUT
    HandlerToFind : I_NotificationHandler;
END_VAR
VAR
    NextHandler : I_NotificationHandler;
    i           : UDINT;
END_VAR
IF HandlerCount < 1 THEN
    RETURN;
END_IF

FOR i := 0 TO HandlerCount - 1 DO
    NextHandler := GetHandler(i);
    IF NextHandler = HandlerToFind THEN
        HandlerInList := TRUE;
    END_IF
END_FOR
END_METHOD

END_FUNCTION_BLOCK

// ---- Classes/Notifications/Notification Handler/T_NotificationHandler.TcPOU
{attribute 'no_explicit_call' := 'do not call this POU directly'}
FUNCTION_BLOCK T_NotificationHandler IMPLEMENTS I_NotificationHandler
VAR
    Args_LocalCopy                      : T_Stream(StreamLength := 4); // Local copy of notification arguments
    Args_PublicCopy                     : T_Stream(StreamLength := 4); // Public copy of notification arguments
    CriticalSection                     : FB_IecCriticalSection;
    NotificationCounter                 : T_Counter;
    QueueingEnabled                     : BOOL;         // if required, set via variable initialisation in instance declaration
    RisingEdge_CriticalSectionInitError : T_RisingEdge; // Sometimes on online change we get CriticalSection.hrInit <> S_OK, so we need to log 1 error message (not every scan!)
    MAX_UNHANDLED_NOTIFICATIONS         : DINT := 10;
END_VAR

PROPERTY Args : I_StreamReader
GET
Args := Args_PublicCopy;
END_GET
END_PROPERTY

METHOD IsRaised : BOOL
VAR
    ByteCount : UDINT;
END_VAR
IF CriticalSection.hrInit = S_OK THEN
	RisingEdge_CriticalSectionInitError.Test(FALSE);
    IF CriticalSection.Enter() THEN           // will block while receiving a notification
        IF NotificationCounter.Value > 0 THEN // at least one unhandled notification to be handled...
            IsRaised := TRUE;

            // get the length of the notification args (this is stored before the args themselves)
            ByteCount := Args_LocalCopy.Read_UDINT();

            // Copy the args for this notification to the public copy of the args, which can be accessed externally...
            Args_PublicCopy.Clear();
            Args_PublicCopy.AppendBytesFromStream(Args_LocalCopy,
                                                  ByteCount);

            NotificationCounter.Dec(); // to keep track of how many notifications remain to be handled

            IF NotificationQueueingEnabled AND NotificationCounter.Value > 0 THEN // more args to be handled (notification raised multiple times since last handled)...
                // advance the read pointer to the args belonging to the next notification (if any)                                      
                Args_LocalCopy.SetReadPosition(Args_LocalCopy.ReadPosition + ByteCount);
            ELSE // clear any unhandled notifications that remain..
				NotificationCounter.Reset();
                Args_LocalCopy.Clear();
            END_IF
        END_IF

        CriticalSection.Leave();
    END_IF
ELSE
	IF RisingEdge_CriticalSectionInitError.Test(TRUE) THEN // send error message only once!
    	F_LogError(Source := 'T_NotificationHandler', Message := 'FB_IEC_CriticalSection not initialised!');
	END_IF
END_IF
END_METHOD

PROPERTY NotificationCount : DINT
GET
NotificationCount := NotificationCounter.Value;
END_GET
END_PROPERTY

PROPERTY NotificationQueueingEnabled : BOOL// Allows notifications to be raised multiple times before being handled sequentially. Make sure all notifications are handled!
GET
NotificationQueueingEnabled := QueueingEnabled;
END_GET
SET
QueueingEnabled := NotificationQueueingEnabled;
END_SET
END_PROPERTY

METHOD RaiseNotification
VAR_INPUT
    NotificationArgs : I_StreamReader;
END_VAR
IF NotificationCounter.Value > MAX_UNHANDLED_NOTIFICATIONS THEN
    // Not much point raising another if they are not being handled...
    RETURN;
END_IF

IF CriticalSection.hrInit = S_OK THEN
	RisingEdge_CriticalSectionInitError.Test(FALSE);
	IF CriticalSection.Enter() THEN
		IF NotificationArgs.WritePosition > 0 THEN // has event arguments..
	
			// Notification args are stored in a local copy using a stream
			// If the notification is raised again before being handled, the newer notification args are just added to the stream
			// The size of the args is stored in the stream before the args themselves so they
			// can be retrieved seperately when the notifications are handled    
	
			Args_LocalCopy.Add_UDINT(NotificationArgs.WritePosition); // length of args is stored first
			Args_LocalCopy.AppendBytesFromStream(StreamToAppend        := NotificationArgs,
												 NumberOfBytesToAppend := NotificationArgs.WritePosition); // followed by args themselves
		END_IF
	
		NotificationCounter.Inc(); // keep track of how many times the notification has been raised, so we can handle each notification seperately
		CriticalSection.Leave();
	END_IF
ELSE
	IF RisingEdge_CriticalSectionInitError.Test(TRUE) THEN // send error message only once!
    	F_LogError(Source := 'T_NotificationHandler', Message := 'FB_IEC_CriticalSection not initialised!');
	END_IF
END_IF
END_METHOD

END_FUNCTION_BLOCK

// ---- Classes/Stream/T_Stream.TcPOU
FUNCTION_BLOCK T_Stream IMPLEMENTS I_StreamWriter, I_StreamReader
VAR

    MemoryManager : FB_DynMem_Manager;
    Buffer        : FB_DynMem_Buffer(ipMemMan := MemoryManager);
    pBuffer       : POINTER TO BYTE;

    _StreamLength  : UDINT := 4;
    _ReadPosition  : UDINT;
    _WritePosition : UDINT;
END_VAR

METHOD PRIVATE _Resize
VAR_INPUT
    NewStreamLength : UDINT;
    Preserve        : BOOL;
END_VAR
Buffer.Resize(nSize     := NewStreamLength,
              bPreserve := Preserve,
              bReset    := TRUE);

_StreamLength := NewStreamLength;
pBuffer       := Buffer.pBuffer;
END_METHOD

METHOD PRIVATE _ResizeIfNecessary
VAR_INPUT
    SpaceRequired : UDINT;
END_VAR
VAR
    NewSize : UDINT;
END_VAR
IF _WritePosition + SpaceRequired > _StreamLength THEN
    _Resize(NewStreamLength := _WritePosition + SpaceRequired,
            Preserve        := TRUE);
END_IF
END_METHOD

METHOD Add_BLOB : I_StreamWriter
VAR_INPUT
    BlobToCopyFrom : ANY;
END_VAR
VAR
    pValue : POINTER TO BYTE;
END_VAR
SetPointerToAlignmentBoundary(Address   := _WritePosition,
                              Alignment := 8);

_ResizeIfNecessary(SpaceRequired := DINT_TO_UDINT(BlobToCopyFrom.diSize));

MEMCPY(destAddr := pBuffer + _WritePosition,
       srcAddr  := BlobToCopyFrom.pValue,
       n        := DINT_TO_UDINT(BlobToCopyFrom.diSize));

_WritePosition := _WritePosition + DINT_TO_UDINT(BlobToCopyFrom.diSize);

Add_BLOB := THIS^;
END_METHOD

METHOD Add_BOOL : I_StreamWriter
VAR_INPUT
    Value : BOOL;
END_VAR
VAR
    pValue : POINTER TO BOOL;
END_VAR
_ResizeIfNecessary(SpaceRequired := SIZEOF(Value));

pValue         := pBuffer + _WritePosition;
pValue^        := Value;
_WritePosition := _WritePosition + SIZEOF(Value);

Add_BOOL := THIS^;
END_METHOD

METHOD Add_BYTE : I_StreamWriter
VAR_INPUT
    Value : BYTE;
END_VAR
VAR
    pValue : POINTER TO BYTE;
END_VAR
_ResizeIfNecessary(SpaceRequired := SIZEOF(Value));

pValue         := pBuffer + _WritePosition;
pValue^        := Value;
_WritePosition := _WritePosition + SIZEOF(Value);

Add_BYTE := THIS^;
END_METHOD

METHOD Add_DATA : I_StreamWriter
VAR_INPUT
    DataAddress : PVOID;
    DataLength  : UDINT;
END_VAR
SetPointerToAlignmentBoundary(Address   := _WritePosition,
                              Alignment := 8);

_ResizeIfNecessary(SpaceRequired := DataLength);

MEMCPY(destAddr := pBuffer + _WritePosition,
       srcAddr  := DataAddress,
       n        := DataLength);

_WritePosition := _WritePosition + DataLength;

Add_DATA := THIS^;
END_METHOD

METHOD Add_DINT : I_StreamWriter
VAR_INPUT
    Value : DINT;
END_VAR
VAR
    pValue : POINTER TO DINT;

    AddressOffset : PVOID;
END_VAR
SetPointerToAlignmentBoundary(Address   := _WritePosition,
                              Alignment := SIZEOF(Value));

_ResizeIfNecessary(SpaceRequired := SIZEOF(Value));

pValue         := pBuffer + _WritePosition;
pValue^        := Value;
_WritePosition := _WritePosition + SIZEOF(Value);

Add_DINT := THIS^;
END_METHOD

METHOD Add_INT : I_StreamWriter
VAR_INPUT
    Value : INT;
END_VAR
VAR
    pValue : POINTER TO INT;
END_VAR
SetPointerToAlignmentBoundary(Address   := _WritePosition,
                              Alignment := SIZEOF(Value));

_ResizeIfNecessary(SpaceRequired := SIZEOF(Value));

pValue         := pBuffer + _WritePosition;
pValue^        := Value;
_WritePosition := _WritePosition + SIZEOF(Value);

Add_INT := THIS^;
END_METHOD

METHOD Add_LINT : I_StreamWriter
VAR_INPUT
    Value : LINT;
END_VAR
VAR
    pValue : POINTER TO LINT;
END_VAR
SetPointerToAlignmentBoundary(Address   := _WritePosition,
                              Alignment := SIZEOF(Value));

_ResizeIfNecessary(SpaceRequired := SIZEOF(Value));

pValue         := pBuffer + _WritePosition;
pValue^        := Value;
_WritePosition := _WritePosition + SIZEOF(Value);

Add_LINT := THIS^;
END_METHOD

METHOD Add_LREAL : I_StreamWriter
VAR_INPUT
    Value : LREAL;
END_VAR
VAR
    pValue : POINTER TO LREAL;
END_VAR
SetPointerToAlignmentBoundary(Address   := _WritePosition,
                              Alignment := SIZEOF(Value));

_ResizeIfNecessary(SpaceRequired := SIZEOF(Value));

pValue         := pBuffer + _WritePosition;
pValue^        := Value;
_WritePosition := _WritePosition + SIZEOF(Value);

Add_LREAL := THIS^;
END_METHOD

METHOD Add_PVOID : I_StreamWriter
VAR_INPUT
    Value : PVOID;
END_VAR
VAR
    pValue : POINTER TO PVOID;
END_VAR
SetPointerToAlignmentBoundary(Address   := _WritePosition,
                              Alignment := SIZEOF(Value));

_ResizeIfNecessary(SpaceRequired := SIZEOF(Value));

pValue         := pBuffer + _WritePosition;
pValue^        := Value;
_WritePosition := _WritePosition + SIZEOF(Value);

Add_PVOID := THIS^;
END_METHOD

METHOD Add_REAL : I_StreamWriter
VAR_INPUT
    Value : REAL;
END_VAR
VAR
    pValue : POINTER TO REAL;
END_VAR
SetPointerToAlignmentBoundary(Address   := _WritePosition,
                              Alignment := SIZEOF(Value));

_ResizeIfNecessary(SpaceRequired := SIZEOF(Value));

pValue         := pBuffer + _WritePosition;
pValue^        := Value;
_WritePosition := _WritePosition + SIZEOF(Value);

Add_REAL := THIS^;
END_METHOD

METHOD Add_STRING : I_StreamWriter // adds any string length as we only store the chars + null byte
VAR_INPUT
    Value : STRING(255);
END_VAR
VAR
    StringSize : UDINT; // number of characters plus the null termination byte
END_VAR
StringSize := INT_TO_UDINT(LEN(Value) + 1);

_ResizeIfNecessary(SpaceRequired := StringSize); // only storing the characters and the null termination byte

MEMCPY(destAddr := pBuffer + _WritePosition,
       srcAddr  := ADR(Value),
       n        := StringSize);

_WritePosition := _WritePosition + StringSize;

Add_STRING := THIS^;
END_METHOD

METHOD Add_STRUCT : I_StreamWriter
VAR_INPUT
    StructureAddress : PVOID;
    StructureLength  : UDINT;
END_VAR
VAR
    pValue : POINTER TO BYTE;
END_VAR
SetPointerToAlignmentBoundary(Address   := _WritePosition,
                              Alignment := 8);

_ResizeIfNecessary(SpaceRequired := StructureLength);

MEMCPY(destAddr := pBuffer + _WritePosition,
       srcAddr  := StructureAddress,
       n        := StructureLength);

_WritePosition := _WritePosition + StructureLength;

Add_STRUCT := THIS^;
END_METHOD

METHOD Add_UDINT : I_StreamWriter
VAR_INPUT
    Value : UDINT;
END_VAR
VAR
    pValue : POINTER TO UDINT;
END_VAR
SetPointerToAlignmentBoundary(Address   := _WritePosition,
                              Alignment := SIZEOF(Value));

_ResizeIfNecessary(SpaceRequired := SIZEOF(Value));

pValue         := pBuffer + _WritePosition;
pValue^        := Value;
_WritePosition := _WritePosition + SIZEOF(Value);

Add_UDINT := THIS^;
END_METHOD

METHOD Add_UINT : I_StreamWriter
VAR_INPUT
    Value : UINT;
END_VAR
VAR
    pValue : POINTER TO UINT;
END_VAR
SetPointerToAlignmentBoundary(Address   := _WritePosition,
                              Alignment := SIZEOF(Value));

_ResizeIfNecessary(SpaceRequired := SIZEOF(Value));

pValue         := pBuffer + _WritePosition;
pValue^        := Value;
_WritePosition := _WritePosition + SIZEOF(Value);

Add_UINT := THIS^;
END_METHOD

METHOD Add_ULINT : I_StreamWriter
VAR_INPUT
    Value : ULINT;
END_VAR
VAR
    pValue : POINTER TO ULINT;
END_VAR
SetPointerToAlignmentBoundary(Address   := _WritePosition,
                              Alignment := SIZEOF(Value));

_ResizeIfNecessary(SpaceRequired := SIZEOF(Value));

pValue         := pBuffer + _WritePosition;
pValue^        := Value;
_WritePosition := _WritePosition + SIZEOF(Value);

Add_ULINT := THIS^;
END_METHOD

METHOD AppendBytesFromStream
VAR_INPUT
    StreamToAppend        : I_StreamReader;
    NumberOfBytesToAppend : UDINT;
END_VAR
VAR

END_VAR
IF StreamToAppend <> 0 THEN

    _ResizeIfNecessary(NumberOfBytesToAppend);

    MEMCPY(destAddr := Buffer.pBuffer + _WritePosition,
           srcAddr  := StreamToAppend.BufferAddress + StreamToAppend.ReadPosition,
           n        := NumberOfBytesToAppend);

    THIS^._WritePosition := THIS^._WritePosition + NumberOfBytesToAppend;
END_IF
END_METHOD

{attribute 'monitoring' := 'call'}
PROPERTY BufferAddress : PVOID
GET
BufferAddress := pBuffer;
END_GET
END_PROPERTY

METHOD Clear : I_StreamWriter
Buffer.Clear();
_ReadPosition  := 0;
_WritePosition := 0;
pBuffer        := Buffer.pBuffer;
Clear          := THIS^;
END_METHOD

METHOD FB_exit : BOOL
VAR_INPUT
    bInCopyCode : BOOL; // if TRUE, the exit method is called for exiting an instance that is copied afterwards (online change).
END_VAR
IF NOT bInCopyCode THEN
    Buffer.DeleteBuffer();
END_IF
END_METHOD

METHOD FB_init : BOOL
VAR_INPUT
    bInitRetains : BOOL; // if TRUE, the retain variables are initialized (warm start / cold start)
    bInCopyCode  : BOOL; // if TRUE, the instance afterwards gets moved into the copy code (online change)
    StreamLength : UDINT;
END_VAR
IF NOT bInCopyCode THEN
    Init(StreamLength);
END_IF
END_METHOD

METHOD GetNextArgTypeId : E_ArgTypeId;
VAR
    pValue : POINTER TO INT;
    Result : INT;
END_VAR
SetPointerToAlignmentBoundary(Address   := _ReadPosition,
                              Alignment := SIZEOF(Result));

IF _ReadPosition + SIZEOF(Result) <= _StreamLength THEN
    pValue           := pBuffer + _ReadPosition;
    Result           := pValue^;
    _ReadPosition    := _ReadPosition + SIZEOF(Result);
    GetNextArgTypeId := Result;
END_IF
END_METHOD

METHOD Init
VAR_INPUT
    StreamLength : UDINT;
END_VAR
IF Buffer.bAvailable THEN
    Buffer.DeleteBuffer();
END_IF

_StreamLength := StreamLength;
Buffer.CreateBuffer(nSize  := _StreamLength,
                    bReset := TRUE);

_ReadPosition  := 0;
_WritePosition := 0;
pBuffer        := Buffer.pBuffer;
END_METHOD

METHOD Read_BLOB
VAR_INPUT
    BlobToCopyTo : ANY;
END_VAR
VAR
    pValue : POINTER TO BYTE;
END_VAR
SetPointerToAlignmentBoundary(Address   := _ReadPosition,
                              Alignment := 8);

IF _ReadPosition + DINT_TO_UDINT(BlobToCopyTo.diSize) <= _StreamLength THEN
    MEMCPY(destAddr := BlobToCopyTo.pValue,
           srcAddr  := pBuffer + _ReadPosition,
           n        := DINT_TO_UDINT(BlobToCopyTo.diSize));

    _ReadPosition := _ReadPosition + DINT_TO_UDINT(BlobToCopyTo.diSize);
END_IF
END_METHOD

METHOD Read_BOOL : BOOL;
VAR
    pValue : POINTER TO BOOL;
    Result : BOOL;
END_VAR
IF _ReadPosition + SIZEOF(Result) <= _StreamLength THEN
    pValue        := pBuffer + _ReadPosition;
    Result        := pValue^;
    _ReadPosition := _ReadPosition + SIZEOF(Result);
    Read_BOOL     := Result;
END_IF
END_METHOD

METHOD Read_BYTE : BYTE;
VAR
    pValue : POINTER TO BYTE;
    Result : BYTE;
END_VAR
IF _ReadPosition + SIZEOF(Result) <= _StreamLength THEN
    pValue        := pBuffer + _ReadPosition;
    Result        := pValue^;
    _ReadPosition := _ReadPosition + SIZEOF(Result);
    Read_BYTE     := Result;
END_IF
END_METHOD

METHOD Read_DATA
VAR_INPUT
    DataAddress : PVOID;
    DataLength  : UDINT;
END_VAR
SetPointerToAlignmentBoundary(Address   := _ReadPosition,
                              Alignment := 8);

IF _ReadPosition + DataLength <= _StreamLength THEN
    MEMCPY(destAddr := DataAddress,
           srcAddr  := pBuffer + _ReadPosition,
           n        := DataLength);

    _ReadPosition := _ReadPosition + DataLength;
END_IF
END_METHOD

METHOD Read_DINT : DINT;
VAR
    pValue : POINTER TO DINT;
    Result : DINT;
END_VAR
SetPointerToAlignmentBoundary(Address   := _ReadPosition,
                              Alignment := SIZEOF(Result));

IF _ReadPosition + SIZEOF(Result) <= _StreamLength THEN
    pValue        := pBuffer + _ReadPosition;
    Result        := pValue^;
    _ReadPosition := _ReadPosition + SIZEOF(Result);
    Read_DINT     := Result;
END_IF
END_METHOD

METHOD Read_INT : INT;
VAR
    pValue : POINTER TO INT;
    Result : INT;
END_VAR
SetPointerToAlignmentBoundary(Address   := _ReadPosition,
                              Alignment := SIZEOF(Result));

IF _ReadPosition + SIZEOF(Result) <= _StreamLength THEN
    pValue        := pBuffer + _ReadPosition;
    Result        := pValue^;
    _ReadPosition := _ReadPosition + SIZEOF(Result);
    Read_INT      := Result;
END_IF
END_METHOD

METHOD Read_LINT : LINT;
VAR
    pValue : POINTER TO LINT;
    Result : LINT;
END_VAR
SetPointerToAlignmentBoundary(Address   := _ReadPosition,
                              Alignment := SIZEOF(Result));

IF _ReadPosition + SIZEOF(Result) <= _StreamLength THEN
    pValue        := pBuffer + _ReadPosition;
    Result        := pValue^;
    _ReadPosition := _ReadPosition + SIZEOF(Result);
    Read_LINT     := Result;
END_IF
END_METHOD

METHOD Read_LREAL : LREAL;
VAR
    pValue : POINTER TO LREAL;
    Result : LREAL;
END_VAR
SetPointerToAlignmentBoundary(Address   := _ReadPosition,
                              Alignment := SIZEOF(Result));

IF _ReadPosition + SIZEOF(Result) <= _StreamLength THEN
    pValue        := pBuffer + _ReadPosition;
    Result        := pValue^;
    _ReadPosition := _ReadPosition + SIZEOF(Result);
    Read_LREAL    := Result;
END_IF
END_METHOD

METHOD Read_PVOID : PVOID;
VAR
    pValue : POINTER TO PVOID;
    Result : PVOID;
END_VAR
SetPointerToAlignmentBoundary(Address   := _ReadPosition,
                              Alignment := SIZEOF(Result));

IF _ReadPosition + SIZEOF(Result) <= _StreamLength THEN
    pValue        := pBuffer + _ReadPosition;
    Result        := pValue^;
    _ReadPosition := _ReadPosition + SIZEOF(Result);
    Read_PVOID    := Result;
END_IF
END_METHOD

METHOD Read_REAL : REAL;
VAR
    pValue : POINTER TO REAL;
    Result : REAL;
END_VAR
SetPointerToAlignmentBoundary(Address   := _ReadPosition,
                              Alignment := SIZEOF(Result));

IF _ReadPosition + SIZEOF(Result) <= _StreamLength THEN
    pValue        := pBuffer + _ReadPosition;
    Result        := pValue^;
    _ReadPosition := _ReadPosition + SIZEOF(Result);
    Read_REAL     := Result;
END_IF
END_METHOD

METHOD Read_STRING : STRING(255);
VAR
    pValue     : POINTER TO STRING(255);
    StringSize : UDINT; // number of characters plus the null termination byte
END_VAR
pValue     := pBuffer + _ReadPosition;
StringSize := INT_TO_UDINT(LEN(pValue^) + 1);
IF _ReadPosition + StringSize <= _StreamLength THEN // end of string is in the buffer, so proceed...
    _ReadPosition := _ReadPosition + StringSize;
    Read_STRING   := pValue^;
END_IF
END_METHOD

METHOD Read_STRUCT
VAR_INPUT
    StructureAddress : PVOID;
    StructureLength  : UDINT;
END_VAR
VAR
    pValue : POINTER TO BYTE;
END_VAR
SetPointerToAlignmentBoundary(Address   := _ReadPosition,
                              Alignment := 8);

IF _ReadPosition + StructureLength <= _StreamLength THEN
    MEMCPY(destAddr := StructureAddress,
           srcAddr  := pBuffer + _ReadPosition,
           n        := StructureLength);

    _ReadPosition := _ReadPosition + StructureLength;
END_IF
END_METHOD

METHOD Read_UDINT : UDINT;
VAR
    pValue : POINTER TO UDINT;
    Result : UDINT;
END_VAR
SetPointerToAlignmentBoundary(Address   := _ReadPosition,
                              Alignment := SIZEOF(Result));

IF _ReadPosition + SIZEOF(Result) <= _StreamLength THEN
    pValue        := pBuffer + _ReadPosition;
    Result        := pValue^;
    _ReadPosition := _ReadPosition + SIZEOF(Result);
    Read_UDINT    := Result;
END_IF
END_METHOD

METHOD Read_UINT : UINT;
VAR
    pValue : POINTER TO UINT;
    Result : UINT;
END_VAR
SetPointerToAlignmentBoundary(Address   := _ReadPosition,
                              Alignment := SIZEOF(Result));

IF _ReadPosition + SIZEOF(Result) <= _StreamLength THEN
    pValue        := pBuffer + _ReadPosition;
    Result        := pValue^;
    _ReadPosition := _ReadPosition + SIZEOF(Result);
    Read_UINT     := Result;
END_IF
END_METHOD

METHOD Read_ULINT : ULINT;
VAR
    pValue : POINTER TO ULINT;
    Result : ULINT;
END_VAR
SetPointerToAlignmentBoundary(Address   := _ReadPosition,
                              Alignment := SIZEOF(Result));

IF _ReadPosition + SIZEOF(Result) <= _StreamLength THEN
    pValue        := pBuffer + _ReadPosition;
    Result        := pValue^;
    _ReadPosition := _ReadPosition + SIZEOF(Result);
    Read_ULINT    := Result;
END_IF
END_METHOD

{attribute 'monitoring' := 'call'}
PROPERTY ReadPosition : UDINT
GET
ReadPosition := _ReadPosition;
END_GET
END_PROPERTY

METHOD SetNextArgTypeId : I_StreamWriter
VAR_INPUT
    Value : E_ArgTypeId;
END_VAR
VAR
    pValue : POINTER TO INT;
END_VAR
SetPointerToAlignmentBoundary(Address   := _WritePosition,
                              Alignment := SIZEOF(Value));

_ResizeIfNecessary(SpaceRequired := SIZEOF(Value));

pValue  := pBuffer + _WritePosition;
pValue^ := Value;
_WritePosition := _WritePosition + SIZEOF(Value);

SetNextArgTypeId := THIS^;
END_METHOD

METHOD SetPointerToAlignmentBoundary
VAR_IN_OUT
    Address : UDINT;
END_VAR
VAR_INPUT
    Alignment : UDINT;
END_VAR
VAR
    AddressOffset : UDINT;
END_VAR
AddressOffset := Address MOD Alignment;
IF AddressOffset > 0 THEN // Write pointer is not at the correct alignment boundary for the type to be added
    Address := Address + (Alignment - AddressOffset);
END_IF
END_METHOD

METHOD SetReadPosition : I_StreamWriter
VAR_INPUT
    Position : UDINT;
END_VAR
IF Position <= _StreamLength THEN
    THIS^._ReadPosition := Position;
END_IF

SetReadPosition := THIS^;
END_METHOD

{attribute 'monitoring' := 'call'}
PROPERTY StreamLength : UDINT
GET
StreamLength := _StreamLength;
END_GET
END_PROPERTY

{attribute 'monitoring' := 'call'}
PROPERTY WritePosition : UDINT
GET
WritePosition := _WritePosition;
END_GET
END_PROPERTY

END_FUNCTION_BLOCK

// ---- Classes/Notifications/Notification/T_Notification.TcPOU
{attribute 'reflection'}
{attribute 'no_explicit_call' := 'do not call this POU directly'}
FUNCTION_BLOCK T_Notification EXTENDS T_Object IMPLEMENTS I_Notification
VAR
    NotificationtHandlers         : T_ListONotificationHandlers(Capacity := 5);
    NotificationArgs              : T_Stream(StreamLength := 8);
    InhibitNoHandlersErrorMessage : BOOL;
END_VAR

METHOD AddNotificationHandler : I_Notification
VAR_INPUT
    Handler : I_NotificationHandler;
END_VAR
NotificationtHandlers.AddHandler(Handler);
AddNotificationHandler := THIS^;
END_METHOD

PROPERTY PUBLIC Args : I_StreamWriter
GET
Args := NotificationArgs;
END_GET
END_PROPERTY

METHOD ClearNotificationHandlers : I_Notification
NotificationtHandlers.Clear();
ClearNotificationHandlers := THIS^;
END_METHOD

METHOD Raise
VAR
    Handler : I_NotificationHandler;
    i       : UDINT;
END_VAR
IF NotificationtHandlers.Count > 0 THEN
    FOR i := 0 TO NotificationtHandlers.Count - 1 DO
        Handler := NotificationtHandlers.GetHandler(i);
        IF Handler <> 0 THEN
            Handler.RaiseNotification(NotificationArgs := NotificationArgs);
        END_IF
    END_FOR
ELSIF NOT InhibitNoHandlersErrorMessage THEN
	InhibitNoHandlersErrorMessage := TRUE; // Only log 1 message
	F_LogWarning(Source := SUPER^._Name, Message := 'Notification has no notification handlers');
	
	_Message.CreateEx(TC_EVENTS.PLC_Exceptions.LogWarning,_Source);
	_Message.ipArguments.AddString('Notification has no notification handlers');
	_Message.Send(0);
	_Message.Release();
END_IF

NotificationArgs.Clear(); // to leave event args empty for next time event is raised
END_METHOD

END_FUNCTION_BLOCK

// ---- Functions/F_LogWarning.TcPOU
FUNCTION F_LogWarning : T_MaxString
VAR_INPUT
    Source  : T_MaxString;
    Message : T_MaxString;
END_VAR
VAR_STAT
    LastMessage        : T_MaxString;
    RepeatMessageCount : UDINT;
END_VAR

IF Message = LastMessage THEN
    F_Inc(RepeatMessageCount);
ELSE
    RepeatMessageCount := 0;
    LastMessage        := Message;
END_IF

IF RepeatMessageCount < 10 THEN // Avoid flooding the Error List...
    ADSLOGSTR(msgCtrlMask := ADSLOG_MSGTYPE_STRING OR ADSLOG_MSGTYPE_WARN OR ADSLOG_MSGTYPE_LOG,
              msgFmtStr   := CONCAT(Source, ' : %s'),
              strArg      := Message);
END_IF

IF RepeatMessageCount = 10 THEN
    ADSLOGSTR(msgCtrlMask := ADSLOG_MSGTYPE_STRING OR ADSLOG_MSGTYPE_ERROR OR ADSLOG_MSGTYPE_LOG,
              msgFmtStr   := 'Log Warnings suspended - too many identical messages!',
              strArg      := '');
END_IF

END_FUNCTION

// ---- Classes/Nullable Base Class/T_NullableBaseClass.TcPOU
FUNCTION_BLOCK ABSTRACT T_NullableBaseClass
VAR
	_Stubbed : BOOL;
END_VAR

METHOD Stub
VAR_INPUT

END_VAR
_Stubbed := TRUE;
END_METHOD

PROPERTY Stubbed : BOOL
GET
Stubbed := _Stubbed;
END_GET
END_PROPERTY

END_FUNCTION_BLOCK

// ---- Functions/F_CompareMem.TcPOU
FUNCTION F_CompareMem : BOOL // TRUE if blocks match
VAR_INPUT
    Source      : ANY;
    Destination : ANY;
END_VAR
VAR
    Result : DINT;
END_VAR

Result := MEMCMP(pBuf1 := Source.pValue,
                 pBuf2 := Destination.pValue,
                 n     := F_DINT_TO_UDINT(Source.diSize));

F_CompareMem := (Result = 0);

END_FUNCTION

// ---- Functions/F_DINT_TO_UDINT.TcPOU
FUNCTION F_DINT_TO_UDINT : UDINT
VAR_INPUT
    value : DINT;
END_VAR
VAR
    inRangeValue : DINT;
END_VAR

inRangeValue    := MAX(0, value); // Only positive values allowe as inputs...
F_DINT_TO_UDINT := DINT_TO_UDINT(inRangeValue);

END_FUNCTION

// ---- Functions/F_CopyMem.TcPOU
FUNCTION F_CopyMem : UDINT
VAR_INPUT
    Source      : ANY;
    Destination : ANY;
END_VAR
VAR
	ByteCount : UDINT;
END_VAR

// Limit the number of bytes to copy to match destination size if less than the source size
ByteCount := F_DINT_TO_UDINT(MIN(Source.diSize, Destination.diSize));

IF ByteCount > 0 THEN
    memcpy(destAddr := Destination.pValue,
           srcAddr  := Source.pValue,
           n        := ByteCount);
END_IF

END_FUNCTION

// ---- Functions/F_DetectOnlineChange.TcPOU
FUNCTION F_DetectOnlineChange : BOOL
VAR_STAT
    StoredOnlineChangeCnt : UDINT := 99;
END_VAR

F_DetectOnlineChange  := (TwinCAT_SystemInfoVarList._AppInfo.OnlineChangeCnt <> StoredOnlineChangeCnt);
StoredOnlineChangeCnt := TwinCAT_SystemInfoVarList._AppInfo.OnlineChangeCnt;

END_FUNCTION

// ---- Functions/F_Dec.TcPOU
FUNCTION F_Dec : BOOL
VAR_INPUT
    in : ANY_INT;
END_VAR
VAR
    pSINT  : POINTER TO SINT;
    pINT   : POINTER TO INT;
    pDINT  : POINTER TO DINT;
    pLINT  : POINTER TO LINT;
    pUSINT : POINTER TO USINT;
    pUINT  : POINTER TO UINT;
    pUDINT : POINTER TO UDINT;
    pULINT : POINTER TO ULINT;
    pBYTE  : POINTER TO BYTE;
    pWORD  : POINTER TO WORD;
    pDWORD : POINTER TO DWORD;
END_VAR

CASE in.TypeClass OF
	// Signed types can go below zero...
    __SYSTEM.TYPE_CLASS.TYPE_SINT:
        pSINT  := in.pValue;
        pSint^ := pSint^ - 1;

    __SYSTEM.TYPE_CLASS.TYPE_INT:
        pINT  := in.pValue;
        pINT^ := pINT^ - 1;

    __SYSTEM.TYPE_CLASS.TYPE_DINT:
        pDINT  := in.pValue;
        pDINT^ := pDINT^ - 1;

    __SYSTEM.TYPE_CLASS.TYPE_LINT:
        pLINT  := in.pValue;
        pLINT^ := pLINT^ - 1;

	// Unsigned types cannot go below zero...
    __SYSTEM.TYPE_CLASS.TYPE_USINT:
        pUSINT := in.pValue;
        IF pUSINT^ > 0 THEN
            pUSINT^ := pUSINT^ - 1;
        END_IF

    __SYSTEM.TYPE_CLASS.TYPE_UINT:
        pUINT  := in.pValue;
        IF pUINT^ > 0 THEN
            pUINT^ := pUINT^ - 1;
        END_IF

    __SYSTEM.TYPE_CLASS.TYPE_UDINT:
        pUDINT  := in.pValue;
        IF pUDINT^ > 0 THEN
            pUDINT^ := pUDINT^ - 1;
        END_IF

    __SYSTEM.TYPE_CLASS.TYPE_ULINT:
        pULINT  := in.pValue;
        IF pULINT^ > 0 THEN
            pULINT^ := pULINT^ - 1;
        END_IF

    __SYSTEM.TYPE_CLASS.TYPE_BYTE:
        pBYTE  := in.pValue;
        IF pBYTE^ > 0 THEN
            pBYTE^ := pBYTE^ - 1;
        END_IF

    __SYSTEM.TYPE_CLASS.TYPE_WORD:
        pWORD  := in.pValue;
        IF pWORD^ > 0 THEN
            pWORD^ := pWORD^ - 1;
        END_IF

    __SYSTEM.TYPE_CLASS.TYPE_DWORD:
        pDWORD  := in.pValue;
        IF pDWORD^ > 0 THEN
            pDWORD^ := pDWORD^ - 1;
        END_IF

END_CASE

END_FUNCTION

// ---- Functions/F_InLimits.TcPOU
FUNCTION F_InLimits : BOOL
VAR_INPUT
    In        : LREAL;
    LowLimit  : LREAL;
    HighLimit : LREAL;
END_VAR

F_InLimits := (In >= LowLimit) AND (In <= HighLimit);

END_FUNCTION

// ---- Functions/F_ErrorIdToString.TcPOU
FUNCTION F_ErrorIdToString : T_MaxString
VAR_INPUT
    ErrorId : UDINT;
END_VAR
VAR
    Result : T_MaxString;
END_VAR

CASE ErrorId OF
    16#0000: Result := 'Error 0x0000 - No error';
    16#0001: Result := 'Error 0x0001 - Internal error';
    16#0002: Result := 'Error 0x0002 - No real-time';
    16#0003: Result := 'Error 0x0003 - Allocation locked – memory error';
    16#0004: Result := 'Error 0x0004 - Mailbox full – the ADS message could not be sent. Reducing the number of ADS messages per cycle will help';
    16#0005: Result := 'Error 0x0005 - Wrong HMSG';
    16#0006: Result := 'Error 0x0006 - Target port not found – ADS server is not started or is not reachable';
    16#0007: Result := 'Error 0x0007 - Target computer not found – AMS route was not found';
    16#0008: Result := 'Error 0x0008 - Unknown command ID';
    16#0009: Result := 'Error 0x0009 - Invalid task ID';
    16#000A: Result := 'Error 0x000A - No IO';
    16#000B: Result := 'Error 0x000B - Unknown AMS command';
    16#000C: Result := 'Error 0x000C - Win32 error';
    16#000D: Result := 'Error 0x000D - Port not connected';
    16#000E: Result := 'Error 0x000E - Invalid AMS length';
    16#000F: Result := 'Error 0x000F - Invalid AMS Net ID';
    16#0010: Result := 'Error 0x0010 - Installation level is too low –TwinCAT 2 license error';
    16#0011: Result := 'Error 0x0011 - No debugging available';
    16#0012: Result := 'Error 0x0012 - Port disabled – TwinCAT system service not started';
    16#0013: Result := 'Error 0x0013 - Port already connected';
    16#0014: Result := 'Error 0x0014 - AMS Sync Win32 error';
    16#0015: Result := 'Error 0x0015 - AMS Sync Timeout';
    16#0016: Result := 'Error 0x0016 - AMS Sync error';
    16#0017: Result := 'Error 0x0017 - No index map for AMS Sync available';
    16#0018: Result := 'Error 0x0018 - Invalid AMS port';
    16#0019: Result := 'Error 0x0019 - No memory';
    16#001A: Result := 'Error 0x001A - TCP send error';
    16#001B: Result := 'Error 0x001B - Host unreachable';
    16#001C: Result := 'Error 0x001C - Invalid AMS fragment';
    16#001D: Result := 'Error 0x001D - TLS send error – secure ADS connection failed';
    16#001E: Result := 'Error 0x001E - Access denied – secure ADS access denied';
    16#0500: Result := 'Error 0x0500 - Locked memory cannot be allocated';
    16#0501: Result := 'Error 0x0501 - The router memory size could not be changed';
    16#0502: Result := 'Error 0x0502 - The mailbox has reached the maximum number of possible messages';
    16#0503: Result := 'Error 0x0503 - The Debug mailbox has reached the maximum number of possible messages';
    16#0504: Result := 'Error 0x0504 - The port type is unknown';
    16#0505: Result := 'Error 0x0505 - The router is not initialized';
    16#0506: Result := 'Error 0x0506 - The port number is already assigned';
    16#0507: Result := 'Error 0x0507 - The port is not registered';
    16#0508: Result := 'Error 0x0508 - The maximum number of ports has been reached';
    16#0509: Result := 'Error 0x0509 - The port is invalid';
    16#050A: Result := 'Error 0x050A - The router is not active';
    16#050B: Result := 'Error 0x050B - The mailbox has reached the maximum number for fragmented messages';
    16#050C: Result := 'Error 0x050C - A fragment timeout has occurred';
    16#050D: Result := 'Error 0x050D - The port is removed';
    16#0700: Result := 'Error 0x0700 - General device error';
    16#0701: Result := 'Error 0x0701 - Service is not supported by the server';
    16#0702: Result := 'Error 0x0702 - Invalid index group';
    16#0703: Result := 'Error 0x0703 - Invalid index offset';
    16#0704: Result := 'Error 0x0704 - Reading or writing not permitted';
    16#0705: Result := 'Error 0x0705 - Parameter size not correct';
    16#0706: Result := 'Error 0x0706 - Invalid data values';
    16#0707: Result := 'Error 0x0707 - Device is not ready to operate';
    16#0708: Result := 'Error 0x0708 - Device is busy';
    16#0709: Result := 'Error 0x0709 - Invalid operating system context. This can result from use of ADS function blocks in different tasks';
    16#070A: Result := 'Error 0x070A - Insufficient memory';
    16#070B: Result := 'Error 0x070B - Invalid parameter values';
    16#070C: Result := 'Error 0x070C - Not found (files, etc...)';
    16#070D: Result := 'Error 0x070D - Syntax error in file or command';
    16#070E: Result := 'Error 0x070E - Objects do not match';
    16#070F: Result := 'Error 0x070F - Object already exists';
    16#0710: Result := 'Error 0x0710 - Symbol not found';
    16#0711: Result := 'Error 0x0711 - Invalid symbol version. This can occur due to an online change - create a new handle';
    16#0712: Result := 'Error 0x0712 - Device (server) is in invalid state';
    16#0713: Result := 'Error 0x0713 - AdsTransMode not supported';
    16#0714: Result := 'Error 0x0714 - Notification handle is invalid';
    16#0715: Result := 'Error 0x0715 - Notification client not registered';
    16#0716: Result := 'Error 0x0716 - No further notification handle available';
    16#0717: Result := 'Error 0x0717 - Notification size too large';
    16#0718: Result := 'Error 0x0718 - Device not initialized';
    16#0719: Result := 'Error 0x0719 - Device has a timeout';
    16#071A: Result := 'Error 0x071A - Interface query failed';
    16#071B: Result := 'Error 0x071B - Wrong interface requested';
    16#071C: Result := 'Error 0x071C - Class ID is invalid';
    16#071D: Result := 'Error 0x071D - Object ID is invalid';
    16#071E: Result := 'Error 0x071E - Request pending';
    16#071F: Result := 'Error 0x071F - Request is aborted';
    16#0720: Result := 'Error 0x0720 - Signal warning';
    16#0721: Result := 'Error 0x0721 - Invalid array index';
    16#0722: Result := 'Error 0x0722 - Symbol not active';
    16#0723: Result := 'Error 0x0723 - Access denied';
    16#0724: Result := 'Error 0x0724 - Missing license';
    16#0725: Result := 'Error 0x0725 - License expired';
    16#0726: Result := 'Error 0x0726 - License exceeded';
    16#0727: Result := 'Error 0x0727 - Invalid license';
    16#0728: Result := 'Error 0x0728 - License problem: System ID is invalid';
    16#0729: Result := 'Error 0x0729 - License not limited in time';
    16#072A: Result := 'Error 0x072A - License problem: Time in the future';
    16#072B: Result := 'Error 0x072B - License period too long';
    16#072C: Result := 'Error 0x072C - Exception at system startup';
    16#072D: Result := 'Error 0x072D - License file read twice';
    16#072E: Result := 'Error 0x072E - Invalid signature';
    16#072F: Result := 'Error 0x072F - Invalid certificate';
    16#0730: Result := 'Error 0x0730 - Public key not known from OEM';
    16#0731: Result := 'Error 0x0731 - License not valid for this system ID';
    16#0732: Result := 'Error 0x0732 - Demo license prohibited';
    16#0733: Result := 'Error 0x0733 - Invalid function ID';
    16#0734: Result := 'Error 0x0734 - Outside the valid range';
    16#0735: Result := 'Error 0x0735 - Invalid alignment';
    16#0736: Result := 'Error 0x0736 - Invalid platform level';
    16#0737: Result := 'Error 0x0737 - Context – forward to passive level';
    16#0738: Result := 'Error 0x0738 - Context – forward to dispatch level';
    16#0739: Result := 'Error 0x0739 - Context – forward to real-time';
    16#0740: Result := 'Error 0x0740 - Client error';
    16#0741: Result := 'Error 0x0741 - Service contains an invalid parameter';
    16#0742: Result := 'Error 0x0742 - Polling list is empty';
    16#0743: Result := 'Error 0x0743 - Var connection already in use';
    16#0744: Result := 'Error 0x0744 - The called ID is already in use';
    16#0745: Result := 'Error 0x0745 - Timeout has occurred –  the remote terminal is not responding in the specified ADS timeout';
    16#0746: Result := 'Error 0x0746 - Error in Win32 subsystem';
    16#0747: Result := 'Error 0x0747 - Invalid client timeout value';
    16#0748: Result := 'Error 0x0748 - Port not open';
    16#0749: Result := 'Error 0x0749 - No AMS address';
    16#0750: Result := 'Error 0x0750 - Internal error in Ads sync';
    16#0751: Result := 'Error 0x0751 - Hash table overflow';
    16#0752: Result := 'Error 0x0752 - Key not found in the table';
    16#0753: Result := 'Error 0x0753 - No symbols in the cache';
    16#0754: Result := 'Error 0x0754 - Invalid response received';
    16#0755: Result := 'Error 0x0755 - Sync Port is locked';
    16#1000: Result := 'Error 0x1000 - Internal error in the real-time system';
    16#1001: Result := 'Error 0x1001 - Timer value is not valid';
    16#1002: Result := 'Error 0x1002 - Task pointer has the invalid value 0 (zero)';
    16#1003: Result := 'Error 0x1003 - Stack pointer has the invalid value 0 (zero)';
    16#1004: Result := 'Error 0x1004 - The request task priority is already assigned';
    16#1005: Result := 'Error 0x1005 - No free TCB (Task Control Block) available. The maximum number of TCBs is 64';
    16#1006: Result := 'Error 0x1006 - No free semaphores available. The maximum number of semaphores is 64';
    16#1007: Result := 'Error 0x1007 - No free space available in the queue. The maximum number of positions in the queue is 64';
    16#100D: Result := 'Error 0x100D - An external synchronization interrupt is already applied';
    16#100E: Result := 'Error 0x100E - No external sync interrupt applied';
    16#100F: Result := 'Error 0x100F - Application of the external synchronization interrupt has failed';
    16#1010: Result := 'Error 0x1010 - Call of a service function in the wrong context';
    16#1017: Result := 'Error 0x1017 - Intel VT-x extension is not supported';
    16#1018: Result := 'Error 0x1018 - Intel VT-x extension is not enabled in the BIOS';
    16#1019: Result := 'Error 0x1019 - Missing function in Intel VT-x extension';
    16#101A: Result := 'Error 0x101A - Activation of Intel VT-x fails';
	
	16#4260: Result := 'Error 0x4260 - Controller enable not present';
	16#4285: Result := 'Error 0x4285 - Invalid accel/decel parameter(s)';          
	16#4286: Result := 'Error 0x4286 - Invalid velocity parameter';                              
	16#42A0: Result := 'Error 0x42A0 - Group/axis consequential error';                                           
	16#4460: Result := 'Error 0x4460 - Target position is below min software position';                      
	16#4461: Result := 'Error 0x4461 - Target position is above max software position';                      
	16#4462: Result := 'Error 0x4462 - Min software position violated';                      
	16#4463: Result := 'Error 0x4463 - Max software position violated';                      
	16#4550: Result := 'Error 0x4550 - Following error limit exceeded';                                           
	16#4650: Result := 'Error 0x4650 - Drive hardware not ready to operate';                                      
	16#4655: Result := 'Error 0x4655 - Invalid IO data for more than n NC cycles';                      

ELSE
    IF (ErrorId AND 16#FFFF0000) > 0 THEN
        Result := F_FormatString1(Format := 'Error 0x%0.8X', F_UDINT(ErrorId));
    ELSE
        Result := F_FormatString1(Format := 'Error 0x%0.4X', F_UDINT(ErrorId));
    END_IF
END_CASE

F_ErrorIdToString := Result;

END_FUNCTION

// ---- Functions/F_LinearInterpolation.TcPOU
FUNCTION F_LinearInterpolation : LREAL
VAR_INPUT
    LowerBound : LREAL;
    UpperBound : LREAL;
    Interval   : LREAL; // Proportion between bounds (0.0 to 1.0)
END_VAR
VAR
END_VAR

IF F_InLimits(Interval, 0.0, 1.0) THEN
    F_LinearInterpolation := LowerBound + Interval * (UpperBound - LowerBound);
END_IF

END_FUNCTION

// ---- Functions/F_LogMessage.TcPOU
FUNCTION F_LogMessage : T_MaxString
VAR_INPUT
    Source  : T_MaxString;
    Message : T_MaxString;
END_VAR
VAR_STAT
    LastMessage        : T_MaxString;
    RepeatMessageCount : UDINT;
END_VAR

IF Message = LastMessage THEN
    F_Inc(RepeatMessageCount);
ELSE
    RepeatMessageCount := 0;
    LastMessage        := Message;
END_IF

IF RepeatMessageCount < 10 THEN // Avoid flooding the Error List...
    ADSLOGSTR(msgCtrlMask := ADSLOG_MSGTYPE_STRING OR ADSLOG_MSGTYPE_HINT OR ADSLOG_MSGTYPE_LOG,
              msgFmtStr   := CONCAT(Source, ' : %s'),
              strArg      := Message);
END_IF

IF RepeatMessageCount = 10 THEN
    ADSLOGSTR(msgCtrlMask := ADSLOG_MSGTYPE_STRING OR ADSLOG_MSGTYPE_ERROR OR ADSLOG_MSGTYPE_LOG,
              msgFmtStr   := 'Log Info suspended - too many identical messages!',
              strArg      := '');
END_IF

END_FUNCTION

// ---- Functions/F_ReadFlag.TcPOU
FUNCTION F_ReadFlag : BOOL // Reads a boolean and clears it if set
VAR_IN_OUT
	Flag : BOOL;
END_VAR

F_ReadFlag := Flag;
Flag       := FALSE;

END_FUNCTION

// ---- Functions/F_TaskTime.TcPOU
FUNCTION F_TaskTime : LREAL
VAR
    TaskIndex : DINT;
END_VAR

TaskIndex := GETCURTASKINDEXEX();
IF TaskIndex > 0 THEN
    F_TaskTime := UDINT_TO_LREAL(TwinCAT_SystemInfoVarList._taskInfo[TaskIndex].CycleTime) * LREAL#1E-7;
END_IF

END_FUNCTION

// ---- Functions/F_NotEqual.TcPOU
FUNCTION F_NotEqual : BOOL
VAR_INPUT
    In1   : LREAL;
    In2   : LREAL;
    Delta : LREAL;
END_VAR
VAR
    Difference : LREAL;
END_VAR

Difference := ABS(In1 - In2);
F_NotEqual := Difference > Delta;

END_FUNCTION

// ---- Functions/F_Toggle.TcPOU
FUNCTION F_Toggle : BOOL
VAR_IN_OUT
	Flag : BOOL;
END_VAR

Flag     := NOT Flag;
F_Toggle := Flag;

END_FUNCTION

// ---- Functions/F_UDINT_TO_DINT.TcPOU
FUNCTION F_UDINT_TO_DINT : DINT
VAR_INPUT
    value : UDINT;
END_VAR
VAR
    inRangeValue : UDINT;
END_VAR

IF value.31 THEN // out of range
    inRangeValue := 16#7FFF_FFFF; // ‭Max DINT = 2147483647‬
ELSE
    inRangeValue := value;
END_IF
F_UDINT_TO_DINT := UDINT_TO_DINT(inRangeValue);

END_FUNCTION

// ---- Functions/F_Equals.TcPOU
FUNCTION F_Equals : BOOL
VAR_INPUT
    In1   : LREAL;
    In2   : LREAL;
    Delta : LREAL;
END_VAR
VAR
    Difference : LREAL;
END_VAR

Difference := ABS(In1 - In2);
F_Equals   := Difference < Delta;

END_FUNCTION

// ---- Functions/F_GetAdsPort.TcPOU
FUNCTION F_GetAdsPort : UINT
VAR
    TaskIndex : DINT;
END_VAR

TaskIndex := GETCURTASKINDEXEX();
IF TaskIndex > 0 THEN
    F_GetAdsPort := TwinCAT_SystemInfoVarList._AppInfo.AdsPort;
END_IF

END_FUNCTION
